LIN {X 0,Y 228.059,Z 101.561,A -85,B 0,C 180,E1 -19963.897,E2 -19963.897} C_VEL
LIN {X 0,Y 228.095,Z 101.553,A -85,B 0,C 180,E1 -19967.544,E2 -19967.544} C_VEL
LIN {X 0,Y 228.307,Z 101.501,A -85,B 0,C 180,E1 -19971.145,E2 -19971.145} C_VEL
LIN {X 0,Y 228.357,Z 101.52,A -85,B 0,C 180,E1 -19972.928,E2 -19972.928} C_VEL
LIN {X 0,Y 228.555,Z 101.482,A -85,B 0,C 180,E1 -19978.237,E2 -19978.237} C_VEL
LIN {X 0,Y 228.554,Z 101.479,A -85,B 0,C 180,E1 -19981.761,E2 -19981.761} C_VEL
LIN {X 0,Y 228.355,Z 101.523,A -85,B 0,C 180,E1 -19987.07,E2 -19987.07} C_VEL
LIN {X 0,Y 228.163,Z 101.521,A -85,B 0,C 180,E1 -19990.649,E2 -19990.649} C_VEL
LIN {X 0,Y 228.065,Z 101.576,A -85,B 0,C 180,E1 -19994.271,E2 -19994.271} C_VEL
LIN {X 0,Y 228.002,Z 101.548,A -85,B 0,C 180,E1 -19997.952,E2 -19997.952} C_VEL
LIN {X 0,Y 227.929,Z 101.59,A -85,B 0,C 180,E1 -20002.328,E2 -20002.328} C_VEL
LIN {X 0,Y 227.94,Z 101.56,A -85,B 0,C 180,E1 -20006.601,E2 -20006.601} C_VEL
LIN {X 0,Y 227.895,Z 101.596,A -85,B 0,C 180,E1 -20010.29,E2 -20010.29} C_VEL
LIN {X 0,Y 227.887,Z 101.574,A -85,B 0,C 180,E1 -20013.717,E2 -20013.717} C_VEL
LIN {X 0,Y 227.869,Z 101.603,A -85,B 0,C 180,E1 -20018.085,E2 -20018.085} C_VEL
LIN {X 0,Y 227.832,Z 101.602,A -85,B 0,C 180,E1 -20022.736,E2 -20022.736} C_VEL
LIN {X 0,Y 227.806,Z 101.544,A -85,B 0,C 180,E1 -20027.257,E2 -20027.257} C_VEL
LIN {X 0,Y 227.867,Z 101.603,A -85,B 0,C 180,E1 -20031.914,E2 -20031.914} C_VEL
LIN {X 0,Y 227.938,Z 101.91,A -85,B 0,C 180,E1 -20032.933,E2 -20032.933} C_VEL
LIN {X 0,Y 228.317,Z 103.201,A -85,B 0,C 180,E1 -20033.245,E2 -20033.245} C_VEL
LIN {X 0,Y 230.06,Z 105.866,A -85,B 0,C 180,E1 -20033.685,E2 -20033.685} C_VEL
LIN {X 0,Y 238.774,Z 120.975,A -85,B 0,C 180,E1 -20035.759,E2 -20035.759} C_VEL
LIN {X 0,Y 245.282,Z 133.413,A -85,B 0,C 180,E1 -20037.221,E2 -20037.221} C_VEL
LIN {X 0,Y 252.662,Z 147.165,A -85,B 0,C 180,E1 -20038.75,E2 -20038.75} C_VEL
LIN {X 0,Y 261.888,Z 160.593,A -85,B 0,C 180,E1 -20040.392,E2 -20040.392} C_VEL
LIN {X 0,Y 272.615,Z 173.13,A -85,B 0,C 180,E1 -20042.043,E2 -20042.043} C_VEL
LIN {X 0,Y 286.64,Z 187.221,A -85,B 0,C 180,E1 -20043.918,E2 -20043.918} C_VEL
LIN {X 0,Y 299.816,Z 198.41,A -85,B 0,C 180,E1 -20045.476,E2 -20045.476} C_VEL
LIN {X 0,Y 307.546,Z 204.743,A -85,B 0,C 180,E1 -20046.479,E2 -20046.479} C_VEL
LIN {X 0,Y 315.788,Z 211.095,A -85,B 0,C 180,E1 -20047.769,E2 -20047.769} C_VEL
LIN {X 0,Y 323.401,Z 216.756,A -85,B 0,C 180,E1 -20049.138,E2 -20049.138} C_VEL
LIN {X 0,Y 331.374,Z 222.775,A -85,B 0,C 180,E1 -20050.773,E2 -20050.773} C_VEL
LIN {X 0,Y 338.305,Z 227.474,A -85,B 0,C 180,E1 -20052.346,E2 -20052.346} C_VEL
LIN {X 0,Y 345.383,Z 232.65,A -85,B 0,C 180,E1 -20054.203,E2 -20054.203} C_VEL
LIN {X 0,Y 348.898,Z 235.005,A -85,B 0,C 180,E1 -20055.211,E2 -20055.211} C_VEL
LIN {X 0,Y 353.812,Z 237.864,A -85,B 0,C 180,E1 -20056.732,E2 -20056.732} C_VEL
LIN {X 0,Y 357.264,Z 240.175,A -85,B 0,C 180,E1 -20057.969,E2 -20057.969} C_VEL
LIN {X 0,Y 361.923,Z 243.575,A -85,B 0,C 180,E1 -20059.935,E2 -20059.935} C_VEL
LIN {X 0,Y 364.411,Z 245.128,A -85,B 0,C 180,E1 -20061.125,E2 -20061.125} C_VEL
LIN {X 0,Y 368.049,Z 247.051,A -85,B 0,C 180,E1 -20063.188,E2 -20063.188} C_VEL
LIN {X 0,Y 369.965,Z 247.87,A -85,B 0,C 180,E1 -20064.55,E2 -20064.55} C_VEL
LIN {X 0,Y 371.214,Z 248.393,A -85,B 0,C 180,E1 -20065.657,E2 -20065.657} C_VEL
LIN {X 0,Y 372.226,Z 248.63,A -85,B 0,C 180,E1 -20066.753,E2 -20066.753} C_VEL
LIN {X 0,Y 372.866,Z 248.985,A -85,B 0,C 180,E1 -20067.84,E2 -20067.84} C_VEL
LIN {X 0,Y 373.208,Z 249.303,A -85,B 0,C 180,E1 -20068.921,E2 -20068.921} C_VEL
LIN {X 0,Y 373.393,Z 249.209,A -85,B 0,C 180,E1 -20070,E2 -20070} C_VEL
LIN {X 0,Y 373.242,Z 249.205,A -85,B 0,C 180,E1 -20071.079,E2 -20071.079} C_VEL
LIN {X 0,Y 372.792,Z 248.918,A -85,B 0,C 180,E1 -20072.349,E2 -20072.349} C_VEL
LIN {X 0,Y 372.235,Z 248.604,A -85,B 0,C 180,E1 -20073.247,E2 -20073.247} C_VEL
LIN {X 0,Y 371.236,Z 248.342,A -85,B 0,C 180,E1 -20074.343,E2 -20074.343} C_VEL
LIN {X 0,Y 369.961,Z 247.901,A -85,B 0,C 180,E1 -20075.45,E2 -20075.45} C_VEL
LIN {X 0,Y 368.054,Z 247.054,A -85,B 0,C 180,E1 -20076.818,E2 -20076.818} C_VEL
LIN {X 0,Y 364.414,Z 245.128,A -85,B 0,C 180,E1 -20078.875,E2 -20078.875} C_VEL
LIN {X 0,Y 361.957,Z 243.542,A -85,B 0,C 180,E1 -20080.064,E2 -20080.064} C_VEL
LIN {X 0,Y 357.625,Z 240.46,A -85,B 0,C 180,E1 -20081.885,E2 -20081.885} C_VEL
LIN {X 0,Y 355.895,Z 239.071,A -85,B 0,C 180,E1 -20082.546,E2 -20082.546} C_VEL
LIN {X 0,Y 351.899,Z 236.864,A -85,B 0,C 180,E1 -20083.866,E2 -20083.866} C_VEL
LIN {X 0,Y 345.467,Z 232.643,A -85,B 0,C 180,E1 -20085.783,E2 -20085.783} C_VEL
LIN {X 0,Y 338.635,Z 227.695,A -85,B 0,C 180,E1 -20087.573,E2 -20087.573} C_VEL
LIN {X 0,Y 331.088,Z 222.551,A -85,B 0,C 180,E1 -20089.286,E2 -20089.286} C_VEL
LIN {X 0,Y 323.395,Z 216.791,A -85,B 0,C 180,E1 -20090.859,E2 -20090.859} C_VEL
LIN {X 0,Y 315.769,Z 211.081,A -85,B 0,C 180,E1 -20092.232,E2 -20092.232} C_VEL
LIN {X 0,Y 307.369,Z 204.614,A -85,B 0,C 180,E1 -20093.547,E2 -20093.547} C_VEL
LIN {X 0,Y 299.628,Z 198.281,A -85,B 0,C 180,E1 -20094.546,E2 -20094.546} C_VEL
LIN {X 0,Y 285.842,Z 186.494,A -85,B 0,C 180,E1 -20096.18,E2 -20096.18} C_VEL
LIN {X 0,Y 271.597,Z 172.061,A -85,B 0,C 180,E1 -20098.104,E2 -20098.104} C_VEL
LIN {X 0,Y 260.976,Z 159.397,A -85,B 0,C 180,E1 -20099.76,E2 -20099.76} C_VEL
LIN {X 0,Y 252.815,Z 147.338,A -85,B 0,C 180,E1 -20101.224,E2 -20101.224} C_VEL
LIN {X 0,Y 245.819,Z 134.485,A -85,B 0,C 180,E1 -20102.662,E2 -20102.662} C_VEL
LIN {X 0,Y 238.898,Z 121.153,A -85,B 0,C 180,E1 -20104.214,E2 -20104.214} C_VEL
LIN {X 0,Y 231.588,Z 108.563,A -85,B 0,C 180,E1 -20105.934,E2 -20105.934} C_VEL
LIN {X 0,Y 229.825,Z 105.609,A -85,B 0,C 180,E1 -20106.368,E2 -20106.368} C_VEL
LIN {X 0,Y 228.192,Z 102.895,A -85,B 0,C 180,E1 -20106.799,E2 -20106.799} C_VEL
LIN {X 0,Y 227.936,Z 101.844,A -85,B 0,C 180,E1 -20107.114,E2 -20107.114} C_VEL
LIN {X 0,Y 227.828,Z 101.552,A -85,B 0,C 180,E1 -20110.376,E2 -20110.376} C_VEL
LIN {X 0,Y 227.829,Z 101.581,A -85,B 0,C 180,E1 -20115.194,E2 -20115.194} C_VEL
LIN {X 0,Y 227.835,Z 101.584,A -85,B 0,C 180,E1 -20119.627,E2 -20119.627} C_VEL
LIN {X 0,Y 227.899,Z 101.579,A -85,B 0,C 180,E1 -20124.133,E2 -20124.133} C_VEL
LIN {X 0,Y 227.867,Z 101.601,A -85,B 0,C 180,E1 -20128.379,E2 -20128.379} C_VEL
LIN {X 0,Y 227.877,Z 101.566,A -85,B 0,C 180,E1 -20132.445,E2 -20132.445} C_VEL
LIN {X 0,Y 227.913,Z 101.595,A -85,B 0,C 180,E1 -20136.368,E2 -20136.368} C_VEL
LIN {X 0,Y 227.941,Z 101.553,A -85,B 0,C 180,E1 -20140.176,E2 -20140.176} C_VEL
LIN {X 0,Y 228.057,Z 101.568,A -85,B 0,C 180,E1 -20143.899,E2 -20143.899} C_VEL
LIN {X 0,Y 228.094,Z 101.554,A -85,B 0,C 180,E1 -20147.545,E2 -20147.545} C_VEL
LIN {X 0,Y 228.306,Z 101.504,A -85,B 0,C 180,E1 -20151.147,E2 -20151.147} C_VEL
LIN {X 0,Y 228.355,Z 101.523,A -85,B 0,C 180,E1 -20152.93,E2 -20152.93} C_VEL
LIN {X 0,Y 228.554,Z 101.479,A -85,B 0,C 180,E1 -20158.239,E2 -20158.239} C_VEL
LIN {X 0,Y 228.555,Z 101.482,A -85,B 0,C 180,E1 -20161.763,E2 -20161.763} C_VEL
LIN {X 0,Y 228.357,Z 101.52,A -85,B 0,C 180,E1 -20167.072,E2 -20167.072} C_VEL
LIN {X 0,Y 228.164,Z 101.52,A -85,B 0,C 180,E1 -20170.651,E2 -20170.651} C_VEL
LIN {X 0,Y 228.066,Z 101.573,A -85,B 0,C 180,E1 -20174.273,E2 -20174.273} C_VEL
LIN {X 0,Y 228.004,Z 101.542,A -85,B 0,C 180,E1 -20177.954,E2 -20177.954} C_VEL
LIN {X 0,Y 227.932,Z 101.589,A -85,B 0,C 180,E1 -20182.33,E2 -20182.33} C_VEL
LIN {X 0,Y 227.943,Z 101.557,A -85,B 0,C 180,E1 -20186.603,E2 -20186.603} C_VEL
LIN {X 0,Y 227.899,Z 101.596,A -85,B 0,C 180,E1 -20190.292,E2 -20190.292} C_VEL
LIN {X 0,Y 227.879,Z 101.572,A -85,B 0,C 180,E1 -20193.721,E2 -20193.721} C_VEL
LIN {X 0,Y 227.846,Z 101.601,A -85,B 0,C 180,E1 -20198.092,E2 -20198.092} C_VEL
LIN {X 0,Y 227.808,Z 101.61,A -85,B 0,C 180,E1 -20202.744,E2 -20202.744} C_VEL
LIN {X 0,Y 227.843,Z 101.602,A -85,B 0,C 180,E1 -20207.505,E2 -20207.505} C_VEL
LIN {X 0,Y 229.24,Z 107.256,A -85,B 0,C 180,E1 -20211.227,E2 -20211.227} C_VEL
LIN {X 0,Y 230.08,Z 111.007,A -85,B 0,C 180,E1 -20213.398,E2 -20213.398} C_VEL
LIN {X 0,Y 231.749,Z 114.816,A -85,B 0,C 180,E1 -20213.952,E2 -20213.952} C_VEL
LIN {X 0,Y 237.983,Z 127.674,A -85,B 0,C 180,E1 -20215.491,E2 -20215.491} C_VEL
LIN {X 0,Y 243.516,Z 140.613,A -85,B 0,C 180,E1 -20216.822,E2 -20216.822} C_VEL
LIN {X 0,Y 247.22,Z 160.789,A -85,B 0,C 180,E1 -20218.055,E2 -20218.055} C_VEL
LIN {X 0,Y 247.03,Z 164.678,A -85,B 0,C 180,E1 -20218.158,E2 -20218.158} C_VEL
LIN {X 0,Y 244.85,Z 170.983,A -85,B 0,C 180,E1 -20218.056,E2 -20218.056} C_VEL
LIN {X 0,Y 242.29,Z 177.323,A -85,B 0,C 180,E1 -20217.898,E2 -20217.898} C_VEL
LIN {X 0,Y 241.549,Z 181.312,A -85,B 0,C 180,E1 -20217.925,E2 -20217.925} C_VEL
LIN {X 0,Y 240.118,Z 217.09,A -85,B 0,C 180,E1 -20218.998,E2 -20218.998} C_VEL
LIN {X 0,Y 239.184,Z 227.774,A -85,B 0,C 180,E1 -20219.503,E2 -20219.503} C_VEL
LIN {X 0,Y 237.783,Z 238.307,A -85,B 0,C 180,E1 -20220.204,E2 -20220.204} C_VEL
LIN {X 0,Y 235.894,Z 250.119,A -85,B 0,C 180,E1 -20221.288,E2 -20221.288} C_VEL
LIN {X 0,Y 233.605,Z 261.513,A -85,B 0,C 180,E1 -20222.691,E2 -20222.691} C_VEL
LIN {X 0,Y 231.127,Z 271.803,A -85,B 0,C 180,E1 -20224.322,E2 -20224.322} C_VEL
LIN {X 0,Y 228.993,Z 280.33,A -85,B 0,C 180,E1 -20226.005,E2 -20226.005} C_VEL
LIN {X 0,Y 227.02,Z 287.546,A -85,B 0,C 180,E1 -20227.714,E2 -20227.714} C_VEL
LIN {X 0,Y 225.012,Z 295.126,A -85,B 0,C 180,E1 -20229.905,E2 -20229.905} C_VEL
LIN {X 0,Y 223.146,Z 301.441,A -85,B 0,C 180,E1 -20232.117,E2 -20232.117} C_VEL
LIN {X 0,Y 221.647,Z 306.704,A -85,B 0,C 180,E1 -20234.364,E2 -20234.364} C_VEL
LIN {X 0,Y 220.182,Z 311.833,A -85,B 0,C 180,E1 -20237.089,E2 -20237.089} C_VEL
LIN {X 0,Y 219.312,Z 315.826,A -85,B 0,C 180,E1 -20239.849,E2 -20239.849} C_VEL
LIN {X 0,Y 218.737,Z 318.78,A -85,B 0,C 180,E1 -20242.616,E2 -20242.616} C_VEL
LIN {X 0,Y 218.501,Z 321.234,A -85,B 0,C 180,E1 -20246.312,E2 -20246.312} C_VEL
LIN {X 0,Y 218.524,Z 321.827,A -85,B 0,C 180,E1 -20248.157,E2 -20248.157} C_VEL
LIN {X 0,Y 218.629,Z 321.985,A -85,B 0,C 180,E1 -20250,E2 -20250} C_VEL
LIN {X 0,Y 218.524,Z 321.827,A -85,B 0,C 180,E1 -20251.843,E2 -20251.843} C_VEL
LIN {X 0,Y 218.484,Z 320.97,A -85,B 0,C 180,E1 -20254.292,E2 -20254.292} C_VEL
LIN {X 0,Y 218.737,Z 318.78,A -85,B 0,C 180,E1 -20257.384,E2 -20257.384} C_VEL
LIN {X 0,Y 219.312,Z 315.826,A -85,B 0,C 180,E1 -20260.151,E2 -20260.151} C_VEL
LIN {X 0,Y 220.182,Z 311.833,A -85,B 0,C 180,E1 -20262.911,E2 -20262.911} C_VEL
LIN {X 0,Y 221.647,Z 306.704,A -85,B 0,C 180,E1 -20265.636,E2 -20265.636} C_VEL
LIN {X 0,Y 223.15,Z 301.441,A -85,B 0,C 180,E1 -20267.883,E2 -20267.883} C_VEL
LIN {X 0,Y 225.051,Z 295.127,A -85,B 0,C 180,E1 -20270.091,E2 -20270.091} C_VEL
LIN {X 0,Y 226.622,Z 289.174,A -85,B 0,C 180,E1 -20271.848,E2 -20271.848} C_VEL
LIN {X 0,Y 228.472,Z 282.248,A -85,B 0,C 180,E1 -20273.571,E2 -20273.571} C_VEL
LIN {X 0,Y 230.659,Z 274.074,A -85,B 0,C 180,E1 -20275.25,E2 -20275.25} C_VEL
LIN {X 0,Y 232.669,Z 265.565,A -85,B 0,C 180,E1 -20276.7,E2 -20276.7} C_VEL
LIN {X 0,Y 234.586,Z 256.854,A -85,B 0,C 180,E1 -20277.912,E2 -20277.912} C_VEL
LIN {X 0,Y 236.222,Z 248.105,A -85,B 0,C 180,E1 -20278.912,E2 -20278.912} C_VEL
LIN {X 0,Y 237.81,Z 238.308,A -85,B 0,C 180,E1 -20279.792,E2 -20279.792} C_VEL
LIN {X 0,Y 239.138,Z 227.8,A -85,B 0,C 180,E1 -20280.502,E2 -20280.502} C_VEL
LIN {X 0,Y 240.011,Z 218.263,A -85,B 0,C 180,E1 -20280.96,E2 -20280.96} C_VEL
LIN {X 0,Y 241.305,Z 187.828,A -85,B 0,C 180,E1 -20281.887,E2 -20281.887} C_VEL
LIN {X 0,Y 241.985,Z 166.994,A -85,B 0,C 180,E1 -20282.502,E2 -20282.502} C_VEL
LIN {X 0,Y 238.111,Z 144.56,A -85,B 0,C 180,E1 -20283.887,E2 -20283.887} C_VEL
LIN {X 0,Y 234.794,Z 136.065,A -85,B 0,C 180,E1 -20284.736,E2 -20284.736} C_VEL
LIN {X 0,Y 228.627,Z 122.664,A -85,B 0,C 180,E1 -20286.316,E2 -20286.316} C_VEL
LIN {X 0,Y 224.217,Z 114.028,A -85,B 0,C 180,E1 -20287.483,E2 -20287.483} C_VEL
LIN {X 0,Y 222.783,Z 110.774,A -85,B 0,C 180,E1 -20288.007,E2 -20288.007} C_VEL
LIN {X 0,Y 221.489,Z 105.488,A -85,B 0,C 180,E1 -20291.331,E2 -20291.331} C_VEL
LIN {X 0,Y 220.777,Z 102.498,A -85,B 0,C 180,E1 -20293.48,E2 -20293.48} C_VEL
LIN {X 0,Y 220.769,Z 102.48,A -85,B 0,C 180,E1 -20298.046,E2 -20298.046} C_VEL
LIN {X 0,Y 220.808,Z 102.462,A -85,B 0,C 180,E1 -20300.462,E2 -20300.462} C_VEL
LIN {X 0,Y 220.803,Z 102.454,A -85,B 0,C 180,E1 -20305.044,E2 -20305.044} C_VEL
LIN {X 0,Y 220.836,Z 102.477,A -85,B 0,C 180,E1 -20309.389,E2 -20309.389} C_VEL
LIN {X 0,Y 220.896,Z 102.434,A -85,B 0,C 180,E1 -20313.549,E2 -20313.549} C_VEL
LIN {X 0,Y 220.88,Z 102.468,A -85,B 0,C 180,E1 -20317.553,E2 -20317.553} C_VEL
LIN {X 0,Y 220.986,Z 102.42,A -85,B 0,C 180,E1 -20322.57,E2 -20322.57} C_VEL
LIN {X 0,Y 221.028,Z 102.44,A -85,B 0,C 180,E1 -20327.138,E2 -20327.138} C_VEL
LIN {X 0,Y 221.238,Z 102.379,A -85,B 0,C 180,E1 -20330.86,E2 -20330.86} C_VEL
LIN {X 0,Y 221.292,Z 102.396,A -85,B 0,C 180,E1 -20332.701,E2 -20332.701} C_VEL
LIN {X 0,Y 221.513,Z 102.358,A -85,B 0,C 180,E1 -20338.181,E2 -20338.181} C_VEL
LIN {X 0,Y 221.512,Z 102.356,A -85,B 0,C 180,E1 -20341.817,E2 -20341.817} C_VEL
LIN {X 0,Y 221.29,Z 102.399,A -85,B 0,C 180,E1 -20347.297,E2 -20347.297} C_VEL
LIN {X 0,Y 221.112,Z 102.401,A -85,B 0,C 180,E1 -20350.993,E2 -20350.993} C_VEL
LIN {X 0,Y 221.016,Z 102.435,A -85,B 0,C 180,E1 -20356.629,E2 -20356.629} C_VEL
LIN {X 0,Y 220.891,Z 102.437,A -85,B 0,C 180,E1 -20360.485,E2 -20360.485} C_VEL
LIN {X 0,Y 220.866,Z 102.467,A -85,B 0,C 180,E1 -20364.434,E2 -20364.434} C_VEL
LIN {X 0,Y 220.825,Z 102.45,A -85,B 0,C 180,E1 -20368.514,E2 -20368.514} C_VEL
LIN {X 0,Y 220.821,Z 102.464,A -85,B 0,C 180,E1 -20372.754,E2 -20372.754} C_VEL
LIN {X 0,Y 220.836,Z 102.478,A -85,B 0,C 180,E1 -20377.287,E2 -20377.287} C_VEL
LIN {X 0,Y 220.784,Z 102.469,A -85,B 0,C 180,E1 -20381.948,E2 -20381.948} C_VEL
LIN {X 0,Y 220.768,Z 102.441,A -85,B 0,C 180,E1 -20385.545,E2 -20385.545} C_VEL
LIN {X 0,Y 220.806,Z 102.44,A -85,B 0,C 180,E1 -20390.463,E2 -20390.463} C_VEL
LIN {X 0,Y 220.874,Z 102.767,A -85,B 0,C 180,E1 -20391.554,E2 -20391.554} C_VEL
LIN {X 0,Y 221.235,Z 104.073,A -85,B 0,C 180,E1 -20391.889,E2 -20391.889} C_VEL
LIN {X 0,Y 222.818,Z 106.604,A -85,B 0,C 180,E1 -20392.324,E2 -20392.324} C_VEL
LIN {X 0,Y 228.374,Z 115.616,A -85,B 0,C 180,E1 -20393.745,E2 -20393.745} C_VEL
LIN {X 0,Y 236.785,Z 130.683,A -85,B 0,C 180,E1 -20395.779,E2 -20395.779} C_VEL
LIN {X 0,Y 246.3,Z 149.277,A -85,B 0,C 180,E1 -20397.912,E2 -20397.912} C_VEL
LIN {X 0,Y 254.449,Z 161.727,A -85,B 0,C 180,E1 -20399.465,E2 -20399.465} C_VEL
LIN {X 0,Y 261.832,Z 171.211,A -85,B 0,C 180,E1 -20400.713,E2 -20400.713} C_VEL
LIN {X 0,Y 273.471,Z 184.014,A -85,B 0,C 180,E1 -20402.455,E2 -20402.455} C_VEL
LIN {X 0,Y 285.366,Z 195.325,A -85,B 0,C 180,E1 -20404.015,E2 -20404.015} C_VEL
LIN {X 0,Y 297.064,Z 205.177,A -85,B 0,C 180,E1 -20405.415,E2 -20405.415} C_VEL
LIN {X 0,Y 305.278,Z 211.84,A -85,B 0,C 180,E1 -20406.528,E2 -20406.528} C_VEL
LIN {X 0,Y 313.149,Z 217.956,A -85,B 0,C 180,E1 -20407.782,E2 -20407.782} C_VEL
LIN {X 0,Y 321.079,Z 223.725,A -85,B 0,C 180,E1 -20409.211,E2 -20409.211} C_VEL
LIN {X 0,Y 329.305,Z 229.918,A -85,B 0,C 180,E1 -20410.923,E2 -20410.923} C_VEL
LIN {X 0,Y 335.922,Z 234.284,A -85,B 0,C 180,E1 -20412.435,E2 -20412.435} C_VEL
LIN {X 0,Y 343.051,Z 239.531,A -85,B 0,C 180,E1 -20414.337,E2 -20414.337} C_VEL
LIN {X 0,Y 348.672,Z 243.15,A -85,B 0,C 180,E1 -20416.003,E2 -20416.003} C_VEL
LIN {X 0,Y 352.897,Z 245.512,A -85,B 0,C 180,E1 -20417.377,E2 -20417.377} C_VEL
LIN {X 0,Y 357.62,Z 249.055,A -85,B 0,C 180,E1 -20419.294,E2 -20419.294} C_VEL
LIN {X 0,Y 361.346,Z 251.519,A -85,B 0,C 180,E1 -20421.049,E2 -20421.049} C_VEL
LIN {X 0,Y 363.544,Z 252.704,A -85,B 0,C 180,E1 -20422.223,E2 -20422.223} C_VEL
LIN {X 0,Y 365.419,Z 253.659,A -85,B 0,C 180,E1 -20423.374,E2 -20423.374} C_VEL
LIN {X 0,Y 367.1,Z 254.352,A -85,B 0,C 180,E1 -20424.568,E2 -20424.568} C_VEL
LIN {X 0,Y 368.285,Z 254.845,A -85,B 0,C 180,E1 -20425.622,E2 -20425.622} C_VEL
LIN {X 0,Y 369.316,Z 255.107,A -85,B 0,C 180,E1 -20426.727,E2 -20426.727} C_VEL
LIN {X 0,Y 369.972,Z 255.445,A -85,B 0,C 180,E1 -20427.823,E2 -20427.823} C_VEL
LIN {X 0,Y 370.311,Z 255.754,A -85,B 0,C 180,E1 -20428.913,E2 -20428.913} C_VEL
LIN {X 0,Y 370.495,Z 255.693,A -85,B 0,C 180,E1 -20430,E2 -20430} C_VEL
LIN {X 0,Y 370.339,Z 255.679,A -85,B 0,C 180,E1 -20431.087,E2 -20431.087} C_VEL
LIN {X 0,Y 369.975,Z 255.415,A -85,B 0,C 180,E1 -20432.177,E2 -20432.177} C_VEL
LIN {X 0,Y 369.326,Z 255.057,A -85,B 0,C 180,E1 -20433.273,E2 -20433.273} C_VEL
LIN {X 0,Y 368.296,Z 254.797,A -85,B 0,C 180,E1 -20434.378,E2 -20434.378} C_VEL
LIN {X 0,Y 366.999,Z 254.346,A -85,B 0,C 180,E1 -20435.494,E2 -20435.494} C_VEL
LIN {X 0,Y 365.433,Z 253.638,A -85,B 0,C 180,E1 -20436.626,E2 -20436.626} C_VEL
LIN {X 0,Y 362.338,Z 252.068,A -85,B 0,C 180,E1 -20438.43,E2 -20438.43} C_VEL
LIN {X 0,Y 358.862,Z 249.906,A -85,B 0,C 180,E1 -20440.152,E2 -20440.152} C_VEL
LIN {X 0,Y 354.957,Z 247.125,A -85,B 0,C 180,E1 -20441.812,E2 -20441.812} C_VEL
LIN {X 0,Y 352.801,Z 245.433,A -85,B 0,C 180,E1 -20442.658,E2 -20442.658} C_VEL
LIN {X 0,Y 347.99,Z 242.708,A -85,B 0,C 180,E1 -20444.212,E2 -20444.212} C_VEL
LIN {X 0,Y 343.044,Z 239.539,A -85,B 0,C 180,E1 -20445.66,E2 -20445.66} C_VEL
LIN {X 0,Y 338.086,Z 235.936,A -85,B 0,C 180,E1 -20447.017,E2 -20447.017} C_VEL
LIN {X 0,Y 330.721,Z 230.874,A -85,B 0,C 180,E1 -20448.764,E2 -20448.764} C_VEL
LIN {X 0,Y 323.251,Z 225.325,A -85,B 0,C 180,E1 -20450.357,E2 -20450.357} C_VEL
LIN {X 0,Y 314.811,Z 219.201,A -85,B 0,C 180,E1 -20451.933,E2 -20451.933} C_VEL
LIN {X 0,Y 306.362,Z 212.683,A -85,B 0,C 180,E1 -20453.309,E2 -20453.309} C_VEL
LIN {X 0,Y 298.371,Z 206.277,A -85,B 0,C 180,E1 -20454.423,E2 -20454.423} C_VEL
LIN {X 0,Y 286.875,Z 196.615,A -85,B 0,C 180,E1 -20455.802,E2 -20455.802} C_VEL
LIN {X 0,Y 276.959,Z 187.471,A -85,B 0,C 180,E1 -20457.067,E2 -20457.067} C_VEL
LIN {X 0,Y 264.203,Z 174.057,A -85,B 0,C 180,E1 -20458.91,E2 -20458.91} C_VEL
LIN {X 0,Y 254.983,Z 162.535,A -85,B 0,C 180,E1 -20460.438,E2 -20460.438} C_VEL
LIN {X 0,Y 246.306,Z 149.26,A -85,B 0,C 180,E1 -20462.088,E2 -20462.088} C_VEL
LIN {X 0,Y 239.106,Z 135.314,A -85,B 0,C 180,E1 -20463.677,E2 -20463.677} C_VEL
LIN {X 0,Y 231.131,Z 120.328,A -85,B 0,C 180,E1 -20465.575,E2 -20465.575} C_VEL
LIN {X 0,Y 224.994,Z 110.1,A -85,B 0,C 180,E1 -20467.109,E2 -20467.109} C_VEL
LIN {X 0,Y 222.657,Z 106.438,A -85,B 0,C 180,E1 -20467.715,E2 -20467.715} C_VEL
LIN {X 0,Y 221.06,Z 103.617,A -85,B 0,C 180,E1 -20468.184,E2 -20468.184} C_VEL
LIN {X 0,Y 220.857,Z 102.683,A -85,B 0,C 180,E1 -20468.516,E2 -20468.516} C_VEL
LIN {X 0,Y 220.768,Z 102.418,A -85,B 0,C 180,E1 -20471.953,E2 -20471.953} C_VEL
LIN {X 0,Y 220.773,Z 102.467,A -85,B 0,C 180,E1 -20475.547,E2 -20475.547} C_VEL
LIN {X 0,Y 220.808,Z 102.464,A -85,B 0,C 180,E1 -20480.465,E2 -20480.465} C_VEL
LIN {X 0,Y 220.832,Z 102.477,A -85,B 0,C 180,E1 -20482.796,E2 -20482.796} C_VEL
LIN {X 0,Y 220.821,Z 102.464,A -85,B 0,C 180,E1 -20487.246,E2 -20487.246} C_VEL
LIN {X 0,Y 220.825,Z 102.45,A -85,B 0,C 180,E1 -20491.486,E2 -20491.486} C_VEL
LIN {X 0,Y 220.866,Z 102.467,A -85,B 0,C 180,E1 -20495.566,E2 -20495.566} C_VEL
LIN {X 0,Y 220.891,Z 102.437,A -85,B 0,C 180,E1 -20499.515,E2 -20499.515} C_VEL
LIN {X 0,Y 221.016,Z 102.435,A -85,B 0,C 180,E1 -20503.371,E2 -20503.371} C_VEL
LIN {X 0,Y 221.112,Z 102.401,A -85,B 0,C 180,E1 -20509.007,E2 -20509.007} C_VEL
LIN {X 0,Y 221.29,Z 102.399,A -85,B 0,C 180,E1 -20512.703,E2 -20512.703} C_VEL
LIN {X 0,Y 221.512,Z 102.356,A -85,B 0,C 180,E1 -20518.183,E2 -20518.183} C_VEL
LIN {X 0,Y 221.513,Z 102.358,A -85,B 0,C 180,E1 -20521.819,E2 -20521.819} C_VEL
LIN {X 0,Y 221.292,Z 102.396,A -85,B 0,C 180,E1 -20527.299,E2 -20527.299} C_VEL
LIN {X 0,Y 221.113,Z 102.4,A -85,B 0,C 180,E1 -20530.995,E2 -20530.995} C_VEL
LIN {X 0,Y 221.018,Z 102.428,A -85,B 0,C 180,E1 -20536.631,E2 -20536.631} C_VEL
LIN {X 0,Y 220.894,Z 102.436,A -85,B 0,C 180,E1 -20540.487,E2 -20540.487} C_VEL
LIN {X 0,Y 220.869,Z 102.461,A -85,B 0,C 180,E1 -20544.436,E2 -20544.436} C_VEL
LIN {X 0,Y 220.829,Z 102.451,A -85,B 0,C 180,E1 -20548.516,E2 -20548.516} C_VEL
LIN {X 0,Y 220.818,Z 102.459,A -85,B 0,C 180,E1 -20552.757,E2 -20552.757} C_VEL
LIN {X 0,Y 220.813,Z 102.481,A -85,B 0,C 180,E1 -20557.279,E2 -20557.279} C_VEL
LIN {X 0,Y 220.796,Z 102.462,A -85,B 0,C 180,E1 -20560.189,E2 -20560.189} C_VEL
LIN {X 0,Y 220.77,Z 102.472,A -85,B 0,C 180,E1 -20564.456,E2 -20564.456} C_VEL
LIN {X 0,Y 220.78,Z 102.537,A -85,B 0,C 180,E1 -20566.645,E2 -20566.645} C_VEL
LIN {X 0,Y 222.642,Z 110.068,A -85,B 0,C 180,E1 -20571.654,E2 -20571.654} C_VEL
LIN {X 0,Y 222.97,Z 111.311,A -85,B 0,C 180,E1 -20572.126,E2 -20572.126} C_VEL
LIN {X 0,Y 229.659,Z 124.833,A -85,B 0,C 180,E1 -20573.953,E2 -20573.953} C_VEL
LIN {X 0,Y 236.147,Z 139.24,A -85,B 0,C 180,E1 -20575.604,E2 -20575.604} C_VEL
LIN {X 0,Y 238.114,Z 144.509,A -85,B 0,C 180,E1 -20576.112,E2 -20576.112} C_VEL
LIN {X 0,Y 241.448,Z 163.621,A -85,B 0,C 180,E1 -20577.301,E2 -20577.301} C_VEL
LIN {X 0,Y 242.072,Z 168.246,A -85,B 0,C 180,E1 -20577.554,E2 -20577.554} C_VEL
LIN {X 0,Y 241.549,Z 181.312,A -85,B 0,C 180,E1 -20577.925,E2 -20577.925} C_VEL
LIN {X 0,Y 240.728,Z 187.162,A -85,B 0,C 180,E1 -20577.999,E2 -20577.999} C_VEL
LIN {X 0,Y 235.124,Z 206.176,A -85,B 0,C 180,E1 -20577.802,E2 -20577.802} C_VEL
LIN {X 0,Y 234.34,Z 212.004,A -85,B 0,C 180,E1 -20577.916,E2 -20577.916} C_VEL
LIN {X 0,Y 233.375,Z 224.851,A -85,B 0,C 180,E1 -20578.461,E2 -20578.461} C_VEL
LIN {X 0,Y 232.06,Z 235.543,A -85,B 0,C 180,E1 -20579.139,E2 -20579.139} C_VEL
LIN {X 0,Y 230.563,Z 244.895,A -85,B 0,C 180,E1 -20579.931,E2 -20579.931} C_VEL
LIN {X 0,Y 228.635,Z 255.031,A -85,B 0,C 180,E1 -20581.044,E2 -20581.044} C_VEL
LIN {X 0,Y 226.646,Z 264.023,A -85,B 0,C 180,E1 -20582.281,E2 -20582.281} C_VEL
LIN {X 0,Y 224.461,Z 272.747,A -85,B 0,C 180,E1 -20583.752,E2 -20583.752} C_VEL
LIN {X 0,Y 222.496,Z 280.139,A -85,B 0,C 180,E1 -20585.258,E2 -20585.258} C_VEL
LIN {X 0,Y 220.429,Z 287.355,A -85,B 0,C 180,E1 -20587.01,E2 -20587.01} C_VEL
LIN {X 0,Y 218.323,Z 294.935,A -85,B 0,C 180,E1 -20589.262,E2 -20589.262} C_VEL
LIN {X 0,Y 216.352,Z 301.249,A -85,B 0,C 180,E1 -20591.535,E2 -20591.535} C_VEL
LIN {X 0,Y 214.779,Z 306.512,A -85,B 0,C 180,E1 -20593.851,E2 -20593.851} C_VEL
LIN {X 0,Y 213.221,Z 311.641,A -85,B 0,C 180,E1 -20596.66,E2 -20596.66} C_VEL
LIN {X 0,Y 212.298,Z 315.635,A -85,B 0,C 180,E1 -20599.509,E2 -20599.509} C_VEL
LIN {X 0,Y 211.671,Z 318.589,A -85,B 0,C 180,E1 -20602.368,E2 -20602.368} C_VEL
LIN {X 0,Y 211.42,Z 321.044,A -85,B 0,C 180,E1 -20606.188,E2 -20606.188} C_VEL
LIN {X 0,Y 211.426,Z 321.636,A -85,B 0,C 180,E1 -20608.095,E2 -20608.095} C_VEL
LIN {X 0,Y 211.545,Z 321.795,A -85,B 0,C 180,E1 -20610,E2 -20610} C_VEL
LIN {X 0,Y 211.426,Z 321.636,A -85,B 0,C 180,E1 -20611.905,E2 -20611.905} C_VEL
LIN {X 0,Y 211.396,Z 320.927,A -85,B 0,C 180,E1 -20614.145,E2 -20614.145} C_VEL
LIN {X 0,Y 211.671,Z 318.589,A -85,B 0,C 180,E1 -20617.632,E2 -20617.632} C_VEL
LIN {X 0,Y 212.298,Z 315.635,A -85,B 0,C 180,E1 -20620.491,E2 -20620.491} C_VEL
LIN {X 0,Y 213.22,Z 311.641,A -85,B 0,C 180,E1 -20623.34,E2 -20623.34} C_VEL
LIN {X 0,Y 214.78,Z 306.512,A -85,B 0,C 180,E1 -20626.149,E2 -20626.149} C_VEL
LIN {X 0,Y 216.357,Z 301.249,A -85,B 0,C 180,E1 -20628.464,E2 -20628.464} C_VEL
LIN {X 0,Y 218.364,Z 294.936,A -85,B 0,C 180,E1 -20630.734,E2 -20630.734} C_VEL
LIN {X 0,Y 220.012,Z 288.983,A -85,B 0,C 180,E1 -20632.54,E2 -20632.54} C_VEL
LIN {X 0,Y 221.978,Z 282.058,A -85,B 0,C 180,E1 -20634.305,E2 -20634.305} C_VEL
LIN {X 0,Y 224.246,Z 273.883,A -85,B 0,C 180,E1 -20636.025,E2 -20636.025} C_VEL
LIN {X 0,Y 226.338,Z 265.375,A -85,B 0,C 180,E1 -20637.509,E2 -20637.509} C_VEL
LIN {X 0,Y 228.331,Z 256.664,A -85,B 0,C 180,E1 -20638.746,E2 -20638.746} C_VEL
LIN {X 0,Y 230.044,Z 247.915,A -85,B 0,C 180,E1 -20639.765,E2 -20639.765} C_VEL
LIN {X 0,Y 231.674,Z 238.117,A -85,B 0,C 180,E1 -20640.665,E2 -20640.665} C_VEL
LIN {X 0,Y 233.033,Z 227.816,A -85,B 0,C 180,E1 -20641.375,E2 -20641.375} C_VEL
LIN {X 0,Y 233.975,Z 217.608,A -85,B 0,C 180,E1 -20641.873,E2 -20641.873} C_VEL
LIN {X 0,Y 235.665,Z 178.995,A -85,B 0,C 180,E1 -20643.052,E2 -20643.052} C_VEL
LIN {X 0,Y 235.976,Z 168.123,A -85,B 0,C 180,E1 -20643.389,E2 -20643.389} C_VEL
LIN {X 0,Y 232.45,Z 147.092,A -85,B 0,C 180,E1 -20644.729,E2 -20644.729} C_VEL
LIN {X 0,Y 228.078,Z 136.184,A -85,B 0,C 180,E1 -20645.902,E2 -20645.902} C_VEL
LIN {X 0,Y 221.785,Z 122.942,A -85,B 0,C 180,E1 -20647.606,E2 -20647.606} C_VEL
LIN {X 0,Y 217.168,Z 114.145,A -85,B 0,C 180,E1 -20648.908,E2 -20648.908} C_VEL
LIN {X 0,Y 215.508,Z 110.625,A -85,B 0,C 180,E1 -20649.508,E2 -20649.508} C_VEL
LIN {X 0,Y 213.928,Z 104.35,A -85,B 0,C 180,E1 -20653.717,E2 -20653.717} C_VEL
LIN {X 0,Y 213.744,Z 103.351,A -85,B 0,C 180,E1 -20654.679,E2 -20654.679} C_VEL
LIN {X 0,Y 213.718,Z 103.346,A -85,B 0,C 180,E1 -20659.142,E2 -20659.142} C_VEL
LIN {X 0,Y 213.746,Z 103.348,A -85,B 0,C 180,E1 -20663.711,E2 -20663.711} C_VEL
LIN {X 0,Y 213.769,Z 103.352,A -85,B 0,C 180,E1 -20668.262,E2 -20668.262} C_VEL
LIN {X 0,Y 213.828,Z 103.313,A -85,B 0,C 180,E1 -20672.602,E2 -20672.602} C_VEL
LIN {X 0,Y 213.854,Z 103.345,A -85,B 0,C 180,E1 -20676.952,E2 -20676.952} C_VEL
LIN {X 0,Y 213.945,Z 103.299,A -85,B 0,C 180,E1 -20682.803,E2 -20682.803} C_VEL
LIN {X 0,Y 213.982,Z 103.322,A -85,B 0,C 180,E1 -20686.707,E2 -20686.707} C_VEL
LIN {X 0,Y 214.169,Z 103.258,A -85,B 0,C 180,E1 -20690.555,E2 -20690.555} C_VEL
LIN {X 0,Y 214.229,Z 103.269,A -85,B 0,C 180,E1 -20692.459,E2 -20692.459} C_VEL
LIN {X 0,Y 214.446,Z 103.238,A -85,B 0,C 180,E1 -20698.121,E2 -20698.121} C_VEL
LIN {X 0,Y 214.547,Z 103.21,A -85,B 0,C 180,E1 -20699.999,E2 -20699.999} C_VEL
LIN {X 0,Y 214.446,Z 103.235,A -85,B 0,C 180,E1 -20701.877,E2 -20701.877} C_VEL
LIN {X 0,Y 214.228,Z 103.273,A -85,B 0,C 180,E1 -20707.539,E2 -20707.539} C_VEL
LIN {X 0,Y 214.045,Z 103.284,A -85,B 0,C 180,E1 -20711.361,E2 -20711.361} C_VEL
LIN {X 0,Y 213.934,Z 103.334,A -85,B 0,C 180,E1 -20715.236,E2 -20715.236} C_VEL
LIN {X 0,Y 213.838,Z 103.306,A -85,B 0,C 180,E1 -20719.186,E2 -20719.186} C_VEL
LIN {X 0,Y 213.846,Z 103.349,A -85,B 0,C 180,E1 -20723.226,E2 -20723.226} C_VEL
LIN {X 0,Y 213.827,Z 103.315,A -85,B 0,C 180,E1 -20727.449,E2 -20727.449} C_VEL
LIN {X 0,Y 213.768,Z 103.356,A -85,B 0,C 180,E1 -20731.736,E2 -20731.736} C_VEL
LIN {X 0,Y 213.752,Z 103.345,A -85,B 0,C 180,E1 -20736.285,E2 -20736.285} C_VEL
LIN {X 0,Y 213.721,Z 103.342,A -85,B 0,C 180,E1 -20741.122,E2 -20741.122} C_VEL
LIN {X 0,Y 213.727,Z 103.361,A -85,B 0,C 180,E1 -20743.672,E2 -20743.672} C_VEL
LIN {X 0,Y 213.7,Z 103.307,A -85,B 0,C 180,E1 -20746.344,E2 -20746.344} C_VEL
LIN {X 0,Y 213.794,Z 103.502,A -85,B 0,C 180,E1 -20749.96,E2 -20749.96} C_VEL
LIN {X 0,Y 214.063,Z 104.635,A -85,B 0,C 180,E1 -20750.372,E2 -20750.372} C_VEL
LIN {X 0,Y 215.627,Z 107.296,A -85,B 0,C 180,E1 -20750.852,E2 -20750.852} C_VEL
LIN {X 0,Y 216.547,Z 108.567,A -85,B 0,C 180,E1 -20751.104,E2 -20751.104} C_VEL
LIN {X 0,Y 223.568,Z 119.926,A -85,B 0,C 180,E1 -20753.001,E2 -20753.001} C_VEL
LIN {X 0,Y 231.862,Z 134.971,A -85,B 0,C 180,E1 -20755.1,E2 -20755.1} C_VEL
LIN {X 0,Y 241.207,Z 153.46,A -85,B 0,C 180,E1 -20757.29,E2 -20757.29} C_VEL
LIN {X 0,Y 249.984,Z 167.005,A -85,B 0,C 180,E1 -20759.028,E2 -20759.028} C_VEL
LIN {X 0,Y 259.189,Z 178.625,A -85,B 0,C 180,E1 -20760.614,E2 -20760.614} C_VEL
LIN {X 0,Y 271.317,Z 191.6,A -85,B 0,C 180,E1 -20762.438,E2 -20762.438} C_VEL
LIN {X 0,Y 282.411,Z 202.002,A -85,B 0,C 180,E1 -20763.923,E2 -20763.923} C_VEL
LIN {X 0,Y 292.263,Z 210.35,A -85,B 0,C 180,E1 -20765.196,E2 -20765.196} C_VEL
LIN {X 0,Y 301.379,Z 217.746,A -85,B 0,C 180,E1 -20766.443,E2 -20766.443} C_VEL
LIN {X 0,Y 308.36,Z 223.145,A -85,B 0,C 180,E1 -20767.534,E2 -20767.534} C_VEL
LIN {X 0,Y 316.304,Z 228.978,A -85,B 0,C 180,E1 -20768.937,E2 -20768.937} C_VEL
LIN {X 0,Y 323.612,Z 234.482,A -85,B 0,C 180,E1 -20770.412,E2 -20770.412} C_VEL
LIN {X 0,Y 330.772,Z 239.383,A -85,B 0,C 180,E1 -20772.006,E2 -20772.006} C_VEL
LIN {X 0,Y 337.806,Z 244.516,A -85,B 0,C 180,E1 -20773.817,E2 -20773.817} C_VEL
LIN {X 0,Y 344.802,Z 249.073,A -85,B 0,C 180,E1 -20775.842,E2 -20775.842} C_VEL
LIN {X 0,Y 349.042,Z 251.434,A -85,B 0,C 180,E1 -20777.204,E2 -20777.204} C_VEL
LIN {X 0,Y 353.971,Z 255.109,A -85,B 0,C 180,E1 -20779.182,E2 -20779.182} C_VEL
LIN {X 0,Y 357.757,Z 257.617,A -85,B 0,C 180,E1 -20780.958,E2 -20780.958} C_VEL
LIN {X 0,Y 361.218,Z 259.483,A -85,B 0,C 180,E1 -20782.868,E2 -20782.868} C_VEL
LIN {X 0,Y 363.568,Z 260.516,A -85,B 0,C 180,E1 -20784.454,E2 -20784.454} C_VEL
LIN {X 0,Y 364.895,Z 261.068,A -85,B 0,C 180,E1 -20785.581,E2 -20785.581} C_VEL
LIN {X 0,Y 366.034,Z 261.398,A -85,B 0,C 180,E1 -20786.766,E2 -20786.766} C_VEL
LIN {X 0,Y 366.653,Z 261.715,A -85,B 0,C 180,E1 -20787.803,E2 -20787.803} C_VEL
LIN {X 0,Y 366.993,Z 262.021,A -85,B 0,C 180,E1 -20788.903,E2 -20788.903} C_VEL
LIN {X 0,Y 367.193,Z 261.964,A -85,B 0,C 180,E1 -20790,E2 -20790} C_VEL
LIN {X 0,Y 367.026,Z 261.949,A -85,B 0,C 180,E1 -20791.097,E2 -20791.097} C_VEL
LIN {X 0,Y 366.659,Z 261.683,A -85,B 0,C 180,E1 -20792.197,E2 -20792.197} C_VEL
LIN {X 0,Y 365.982,Z 261.335,A -85,B 0,C 180,E1 -20793.303,E2 -20793.303} C_VEL
LIN {X 0,Y 364.893,Z 261.042,A -85,B 0,C 180,E1 -20794.419,E2 -20794.419} C_VEL
LIN {X 0,Y 363.54,Z 260.529,A -85,B 0,C 180,E1 -20795.547,E2 -20795.547} C_VEL
LIN {X 0,Y 361.227,Z 259.479,A -85,B 0,C 180,E1 -20797.144,E2 -20797.144} C_VEL
LIN {X 0,Y 357.751,Z 257.601,A -85,B 0,C 180,E1 -20799.042,E2 -20799.042} C_VEL
LIN {X 0,Y 355.228,Z 255.977,A -85,B 0,C 180,E1 -20800.257,E2 -20800.257} C_VEL
LIN {X 0,Y 351.742,Z 253.523,A -85,B 0,C 180,E1 -20801.753,E2 -20801.753} C_VEL
LIN {X 0,Y 349.05,Z 251.469,A -85,B 0,C 180,E1 -20802.796,E2 -20802.796} C_VEL
LIN {X 0,Y 344.788,Z 249.054,A -85,B 0,C 180,E1 -20804.158,E2 -20804.158} C_VEL
LIN {X 0,Y 339.943,Z 245.947,A -85,B 0,C 180,E1 -20805.591,E2 -20805.591} C_VEL
LIN {X 0,Y 334.315,Z 241.909,A -85,B 0,C 180,E1 -20807.116,E2 -20807.116} C_VEL
LIN {X 0,Y 326.823,Z 236.779,A -85,B 0,C 180,E1 -20808.886,E2 -20808.886} C_VEL
LIN {X 0,Y 319.715,Z 231.508,A -85,B 0,C 180,E1 -20810.401,E2 -20810.401} C_VEL
LIN {X 0,Y 310.855,Z 225.076,A -85,B 0,C 180,E1 -20812.038,E2 -20812.038} C_VEL
LIN {X 0,Y 301.976,Z 218.197,A -85,B 0,C 180,E1 -20813.473,E2 -20813.473} C_VEL
LIN {X 0,Y 293.186,Z 211.137,A -85,B 0,C 180,E1 -20814.682,E2 -20814.682} C_VEL
LIN {X 0,Y 282.604,Z 202.144,A -85,B 0,C 180,E1 -20816.056,E2 -20816.056} C_VEL
LIN {X 0,Y 273.016,Z 193.289,A -85,B 0,C 180,E1 -20817.325,E2 -20817.325} C_VEL
LIN {X 0,Y 259.716,Z 179.264,A -85,B 0,C 180,E1 -20819.3,E2 -20819.3} C_VEL
LIN {X 0,Y 250.278,Z 167.434,A -85,B 0,C 180,E1 -20820.917,E2 -20820.917} C_VEL
LIN {X 0,Y 241.047,Z 153.175,A -85,B 0,C 180,E1 -20822.745,E2 -20822.745} C_VEL
LIN {X 0,Y 229.278,Z 130.087,A -85,B 0,C 180,E1 -20825.539,E2 -20825.539} C_VEL
LIN {X 0,Y 221.074,Z 115.603,A -85,B 0,C 180,E1 -20827.665,E2 -20827.665} C_VEL
LIN {X 0,Y 216.462,Z 108.372,A -85,B 0,C 180,E1 -20828.922,E2 -20828.922} C_VEL
LIN {X 0,Y 214.249,Z 105.123,A -85,B 0,C 180,E1 -20829.553,E2 -20829.553} C_VEL
LIN {X 0,Y 213.829,Z 103.768,A -85,B 0,C 180,E1 -20829.871,E2 -20829.871} C_VEL
LIN {X 0,Y 213.743,Z 103.361,A -85,B 0,C 180,E1 -20830.403,E2 -20830.403} C_VEL
LIN {X 0,Y 213.7,Z 103.307,A -85,B 0,C 180,E1 -20833.68,E2 -20833.68} C_VEL
LIN {X 0,Y 213.727,Z 103.361,A -85,B 0,C 180,E1 -20836.338,E2 -20836.338} C_VEL
LIN {X 0,Y 213.735,Z 103.355,A -85,B 0,C 180,E1 -20841.337,E2 -20841.337} C_VEL
LIN {X 0,Y 213.766,Z 103.331,A -85,B 0,C 180,E1 -20846.021,E2 -20846.021} C_VEL
LIN {X 0,Y 213.758,Z 103.344,A -85,B 0,C 180,E1 -20850.452,E2 -20850.452} C_VEL
LIN {X 0,Y 213.799,Z 103.333,A -85,B 0,C 180,E1 -20854.703,E2 -20854.703} C_VEL
LIN {X 0,Y 213.812,Z 103.328,A -85,B 0,C 180,E1 -20858.804,E2 -20858.804} C_VEL
LIN {X 0,Y 213.943,Z 103.306,A -85,B 0,C 180,E1 -20862.805,E2 -20862.805} C_VEL
LIN {X 0,Y 213.981,Z 103.324,A -85,B 0,C 180,E1 -20866.709,E2 -20866.709} C_VEL
LIN {X 0,Y 214.167,Z 103.26,A -85,B 0,C 180,E1 -20870.557,E2 -20870.557} C_VEL
LIN {X 0,Y 214.228,Z 103.273,A -85,B 0,C 180,E1 -20872.461,E2 -20872.461} C_VEL
LIN {X 0,Y 214.446,Z 103.235,A -85,B 0,C 180,E1 -20878.123,E2 -20878.123} C_VEL
LIN {X 0,Y 214.547,Z 103.21,A -85,B 0,C 180,E1 -20880.001,E2 -20880.001} C_VEL
LIN {X 0,Y 214.446,Z 103.238,A -85,B 0,C 180,E1 -20881.879,E2 -20881.879} C_VEL
LIN {X 0,Y 214.229,Z 103.269,A -85,B 0,C 180,E1 -20887.541,E2 -20887.541} C_VEL
LIN {X 0,Y 214.046,Z 103.284,A -85,B 0,C 180,E1 -20891.363,E2 -20891.363} C_VEL
LIN {X 0,Y 213.936,Z 103.329,A -85,B 0,C 180,E1 -20895.238,E2 -20895.238} C_VEL
LIN {X 0,Y 213.841,Z 103.302,A -85,B 0,C 180,E1 -20899.188,E2 -20899.188} C_VEL
LIN {X 0,Y 213.849,Z 103.346,A -85,B 0,C 180,E1 -20903.228,E2 -20903.228} C_VEL
LIN {X 0,Y 213.831,Z 103.313,A -85,B 0,C 180,E1 -20907.451,E2 -20907.451} C_VEL
LIN {X 0,Y 213.769,Z 103.352,A -85,B 0,C 180,E1 -20911.738,E2 -20911.738} C_VEL
LIN {X 0,Y 213.746,Z 103.348,A -85,B 0,C 180,E1 -20916.289,E2 -20916.289} C_VEL
LIN {X 0,Y 213.713,Z 103.348,A -85,B 0,C 180,E1 -20921.126,E2 -20921.126} C_VEL
LIN {X 0,Y 213.743,Z 103.496,A -85,B 0,C 180,E1 -20925.657,E2 -20925.657} C_VEL
LIN {X 0,Y 215.27,Z 109.884,A -85,B 0,C 180,E1 -20930.114,E2 -20930.114} C_VEL
LIN {X 0,Y 215.572,Z 110.882,A -85,B 0,C 180,E1 -20930.563,E2 -20930.563} C_VEL
LIN {X 0,Y 217.783,Z 114.99,A -85,B 0,C 180,E1 -20931.256,E2 -20931.256} C_VEL
LIN {X 0,Y 224.757,Z 129.028,A -85,B 0,C 180,E1 -20933.209,E2 -20933.209} C_VEL
LIN {X 0,Y 231.771,Z 145.022,A -85,B 0,C 180,E1 -20935.079,E2 -20935.079} C_VEL
LIN {X 0,Y 232.771,Z 148.79,A -85,B 0,C 180,E1 -20935.388,E2 -20935.388} C_VEL
LIN {X 0,Y 235.575,Z 165.515,A -85,B 0,C 180,E1 -20936.454,E2 -20936.454} C_VEL
LIN {X 0,Y 236.065,Z 169.522,A -85,B 0,C 180,E1 -20936.675,E2 -20936.675} C_VEL
LIN {X 0,Y 234.34,Z 212.004,A -85,B 0,C 180,E1 -20937.916,E2 -20937.916} C_VEL
LIN {X 0,Y 233.481,Z 217.828,A -85,B 0,C 180,E1 -20938.054,E2 -20938.054} C_VEL
LIN {X 0,Y 230.251,Z 227.215,A -85,B 0,C 180,E1 -20938.127,E2 -20938.127} C_VEL
LIN {X 0,Y 226.557,Z 236.391,A -85,B 0,C 180,E1 -20938.353,E2 -20938.353} C_VEL
LIN {X 0,Y 224.986,Z 241.883,A -85,B 0,C 180,E1 -20938.741,E2 -20938.741} C_VEL
LIN {X 0,Y 222.779,Z 253.209,A -85,B 0,C 180,E1 -20939.947,E2 -20939.947} C_VEL
LIN {X 0,Y 220.738,Z 262.482,A -85,B 0,C 180,E1 -20941.213,E2 -20941.213} C_VEL
LIN {X 0,Y 218.423,Z 271.422,A -85,B 0,C 180,E1 -20942.709,E2 -20942.709} C_VEL
LIN {X 0,Y 216.055,Z 279.948,A -85,B 0,C 180,E1 -20944.469,E2 -20944.469} C_VEL
LIN {X 0,Y 213.903,Z 287.164,A -85,B 0,C 180,E1 -20946.266,E2 -20946.266} C_VEL
LIN {X 0,Y 212.011,Z 293.503,A -85,B 0,C 180,E1 -20948.155,E2 -20948.155} C_VEL
LIN {X 0,Y 210.01,Z 299.903,A -85,B 0,C 180,E1 -20950.449,E2 -20950.449} C_VEL
LIN {X 0,Y 208.63,Z 304.406,A -85,B 0,C 180,E1 -20952.351,E2 -20952.351} C_VEL
LIN {X 0,Y 206.788,Z 309.896,A -85,B 0,C 180,E1 -20955.232,E2 -20955.232} C_VEL
LIN {X 0,Y 205.567,Z 314.224,A -85,B 0,C 180,E1 -20958.163,E2 -20958.163} C_VEL
LIN {X 0,Y 205.022,Z 316.595,A -85,B 0,C 180,E1 -20960.131,E2 -20960.131} C_VEL
LIN {X 0,Y 204.627,Z 318.398,A -85,B 0,C 180,E1 -20962.104,E2 -20962.104} C_VEL
LIN {X 0,Y 204.339,Z 320.853,A -85,B 0,C 180,E1 -20966.056,E2 -20966.056} C_VEL
LIN {X 0,Y 204.332,Z 321.446,A -85,B 0,C 180,E1 -20968.029,E2 -20968.029} C_VEL
LIN {X 0,Y 204.443,Z 321.604,A -85,B 0,C 180,E1 -20970,E2 -20970} C_VEL
LIN {X 0,Y 204.331,Z 321.446,A -85,B 0,C 180,E1 -20971.971,E2 -20971.971} C_VEL
LIN {X 0,Y 204.299,Z 320.852,A -85,B 0,C 180,E1 -20973.945,E2 -20973.945} C_VEL
LIN {X 0,Y 204.627,Z 318.398,A -85,B 0,C 180,E1 -20977.896,E2 -20977.896} C_VEL
LIN {X 0,Y 205.276,Z 315.443,A -85,B 0,C 180,E1 -20980.854,E2 -20980.854} C_VEL
LIN {X 0,Y 206.277,Z 311.449,A -85,B 0,C 180,E1 -20983.798,E2 -20983.798} C_VEL
LIN {X 0,Y 207.941,Z 306.321,A -85,B 0,C 180,E1 -20986.695,E2 -20986.695} C_VEL
LIN {X 0,Y 209.606,Z 301.058,A -85,B 0,C 180,E1 -20989.081,E2 -20989.081} C_VEL
LIN {X 0,Y 211.722,Z 294.745,A -85,B 0,C 180,E1 -20991.416,E2 -20991.416} C_VEL
LIN {X 0,Y 213.442,Z 288.792,A -85,B 0,C 180,E1 -20993.274,E2 -20993.274} C_VEL
LIN {X 0,Y 215.502,Z 281.866,A -85,B 0,C 180,E1 -20995.085,E2 -20995.085} C_VEL
LIN {X 0,Y 217.866,Z 273.692,A -85,B 0,C 180,E1 -20996.847,E2 -20996.847} C_VEL
LIN {X 0,Y 220.071,Z 265.184,A -85,B 0,C 180,E1 -20998.362,E2 -20998.362} C_VEL
LIN {X 0,Y 222.116,Z 256.473,A -85,B 0,C 180,E1 -20999.63,E2 -20999.63} C_VEL
LIN {X 0,Y 223.909,Z 247.725,A -85,B 0,C 180,E1 -21000.667,E2 -21000.667} C_VEL
LIN {X 0,Y 225.595,Z 237.927,A -85,B 0,C 180,E1 -21001.585,E2 -21001.585} C_VEL
LIN {X 0,Y 226.992,Z 227.83,A -85,B 0,C 180,E1 -21002.295,E2 -21002.295} C_VEL
LIN {X 0,Y 228.008,Z 217.013,A -85,B 0,C 180,E1 -21002.831,E2 -21002.831} C_VEL
LIN {X 0,Y 230.117,Z 170.352,A -85,B 0,C 180,E1 -21004.267,E2 -21004.267} C_VEL
LIN {X 0,Y 228.143,Z 157.163,A -85,B 0,C 180,E1 -21005.097,E2 -21005.097} C_VEL
LIN {X 0,Y 226.561,Z 148.723,A -85,B 0,C 180,E1 -21005.698,E2 -21005.698} C_VEL
LIN {X 0,Y 220.566,Z 134.691,A -85,B 0,C 180,E1 -21007.377,E2 -21007.377} C_VEL
LIN {X 0,Y 214.128,Z 121.555,A -85,B 0,C 180,E1 -21009.249,E2 -21009.249} C_VEL
LIN {X 0,Y 210.156,Z 114.327,A -85,B 0,C 180,E1 -21010.45,E2 -21010.45} C_VEL
LIN {X 0,Y 208.186,Z 110.418,A -85,B 0,C 180,E1 -21011.181,E2 -21011.181} C_VEL
LIN {X 0,Y 207.273,Z 106.889,A -85,B 0,C 180,E1 -21013.575,E2 -21013.575} C_VEL
LIN {X 0,Y 206.664,Z 104.243,A -85,B 0,C 180,E1 -21015.728,E2 -21015.728} C_VEL
LIN {X 0,Y 206.662,Z 104.222,A -85,B 0,C 180,E1 -21019.748,E2 -21019.748} C_VEL
LIN {X 0,Y 206.701,Z 104.212,A -85,B 0,C 180,E1 -21024.688,E2 -21024.688} C_VEL
LIN {X 0,Y 206.709,Z 104.237,A -85,B 0,C 180,E1 -21029.336,E2 -21029.336} C_VEL
LIN {X 0,Y 206.734,Z 104.198,A -85,B 0,C 180,E1 -21033.771,E2 -21033.771} C_VEL
LIN {X 0,Y 206.76,Z 104.219,A -85,B 0,C 180,E1 -21038.042,E2 -21038.042} C_VEL
LIN {X 0,Y 206.875,Z 104.172,A -85,B 0,C 180,E1 -21042.196,E2 -21042.196} C_VEL
LIN {X 0,Y 206.916,Z 104.205,A -85,B 0,C 180,E1 -21046.245,E2 -21046.245} C_VEL
LIN {X 0,Y 207.107,Z 104.136,A -85,B 0,C 180,E1 -21050.23,E2 -21050.23} C_VEL
LIN {X 0,Y 207.17,Z 104.143,A -85,B 0,C 180,E1 -21052.2,E2 -21052.2} C_VEL
LIN {X 0,Y 207.383,Z 104.118,A -85,B 0,C 180,E1 -21058.057,E2 -21058.057} C_VEL
LIN {X 0,Y 207.512,Z 104.085,A -85,B 0,C 180,E1 -21059.999,E2 -21059.999} C_VEL
LIN {X 0,Y 207.383,Z 104.115,A -85,B 0,C 180,E1 -21061.941,E2 -21061.941} C_VEL
LIN {X 0,Y 207.168,Z 104.146,A -85,B 0,C 180,E1 -21067.798,E2 -21067.798} C_VEL
LIN {X 0,Y 206.982,Z 104.168,A -85,B 0,C 180,E1 -21071.754,E2 -21071.754} C_VEL
LIN {X 0,Y 206.868,Z 104.21,A -85,B 0,C 180,E1 -21075.77,E2 -21075.77} C_VEL
LIN {X 0,Y 206.782,Z 104.187,A -85,B 0,C 180,E1 -21079.868,E2 -21079.868} C_VEL
LIN {X 0,Y 206.762,Z 104.228,A -85,B 0,C 180,E1 -21084.071,E2 -21084.071} C_VEL
LIN {X 0,Y 206.735,Z 104.203,A -85,B 0,C 180,E1 -21088.419,E2 -21088.419} C_VEL
LIN {X 0,Y 206.703,Z 104.218,A -85,B 0,C 180,E1 -21092.955,E2 -21092.955} C_VEL
LIN {X 0,Y 206.72,Z 104.21,A -85,B 0,C 180,E1 -21095.319,E2 -21095.319} C_VEL
LIN {X 0,Y 206.668,Z 104.22,A -85,B 0,C 180,E1 -21100.248,E2 -21100.248} C_VEL
LIN {X 0,Y 206.645,Z 104.222,A -85,B 0,C 180,E1 -21104.422,E2 -21104.422} C_VEL
LIN {X 0,Y 206.685,Z 104.418,A -85,B 0,C 180,E1 -21108.335,E2 -21108.335} C_VEL
LIN {X 0,Y 206.992,Z 105.58,A -85,B 0,C 180,E1 -21108.767,E2 -21108.767} C_VEL
LIN {X 0,Y 208.656,Z 108.294,A -85,B 0,C 180,E1 -21109.309,E2 -21109.309} C_VEL
LIN {X 0,Y 209.686,Z 109.632,A -85,B 0,C 180,E1 -21109.611,E2 -21109.611} C_VEL
LIN {X 0,Y 218.531,Z 123.671,A -85,B 0,C 180,E1 -21112.145,E2 -21112.145} C_VEL
LIN {X 0,Y 227.217,Z 139.779,A -85,B 0,C 180,E1 -21114.457,E2 -21114.457} C_VEL
LIN {X 0,Y 236.095,Z 157.549,A -85,B 0,C 180,E1 -21116.63,E2 -21116.63} C_VEL
LIN {X 0,Y 244.313,Z 170.447,A -85,B 0,C 180,E1 -21118.337,E2 -21118.337} C_VEL
LIN {X 0,Y 252.332,Z 180.968,A -85,B 0,C 180,E1 -21119.802,E2 -21119.802} C_VEL
LIN {X 0,Y 264.524,Z 194.547,A -85,B 0,C 180,E1 -21121.751,E2 -21121.751} C_VEL
LIN {X 0,Y 276.26,Z 205.847,A -85,B 0,C 180,E1 -21123.425,E2 -21123.425} C_VEL
LIN {X 0,Y 286.635,Z 214.904,A -85,B 0,C 180,E1 -21124.912,E2 -21124.912} C_VEL
LIN {X 0,Y 296.848,Z 223.203,A -85,B 0,C 180,E1 -21126.368,E2 -21126.368} C_VEL
LIN {X 0,Y 304.245,Z 228.93,A -85,B 0,C 180,E1 -21127.514,E2 -21127.514} C_VEL
LIN {X 0,Y 312.027,Z 234.642,A -85,B 0,C 180,E1 -21128.877,E2 -21128.877} C_VEL
LIN {X 0,Y 318.782,Z 239.715,A -85,B 0,C 180,E1 -21130.228,E2 -21130.228} C_VEL
LIN {X 0,Y 325.65,Z 244.491,A -85,B 0,C 180,E1 -21131.727,E2 -21131.727} C_VEL
LIN {X 0,Y 330.757,Z 248.061,A -85,B 0,C 180,E1 -21132.971,E2 -21132.971} C_VEL
LIN {X 0,Y 335.747,Z 251.727,A -85,B 0,C 180,E1 -21134.34,E2 -21134.34} C_VEL
LIN {X 0,Y 340.733,Z 254.903,A -85,B 0,C 180,E1 -21135.792,E2 -21135.792} C_VEL
LIN {X 0,Y 345.686,Z 257.752,A -85,B 0,C 180,E1 -21137.383,E2 -21137.383} C_VEL
LIN {X 0,Y 350.427,Z 261.283,A -85,B 0,C 180,E1 -21139.329,E2 -21139.329} C_VEL
LIN {X 0,Y 355.177,Z 264.281,A -85,B 0,C 180,E1 -21141.631,E2 -21141.631} C_VEL
LIN {X 0,Y 357.948,Z 265.727,A -85,B 0,C 180,E1 -21143.235,E2 -21143.235} C_VEL
LIN {X 0,Y 359.991,Z 266.594,A -85,B 0,C 180,E1 -21144.651,E2 -21144.651} C_VEL
LIN {X 0,Y 362.108,Z 267.339,A -85,B 0,C 180,E1 -21146.662,E2 -21146.662} C_VEL
LIN {X 0,Y 362.817,Z 267.672,A -85,B 0,C 180,E1 -21147.78,E2 -21147.78} C_VEL
LIN {X 0,Y 363.155,Z 267.985,A -85,B 0,C 180,E1 -21148.891,E2 -21148.891} C_VEL
LIN {X 0,Y 363.365,Z 267.945,A -85,B 0,C 180,E1 -21150,E2 -21150} C_VEL
LIN {X 0,Y 363.197,Z 267.911,A -85,B 0,C 180,E1 -21151.109,E2 -21151.109} C_VEL
LIN {X 0,Y 362.823,Z 267.639,A -85,B 0,C 180,E1 -21152.22,E2 -21152.22} C_VEL
LIN {X 0,Y 362.119,Z 267.288,A -85,B 0,C 180,E1 -21153.338,E2 -21153.338} C_VEL
LIN {X 0,Y 359.983,Z 266.604,A -85,B 0,C 180,E1 -21155.336,E2 -21155.336} C_VEL
LIN {X 0,Y 357.943,Z 265.704,A -85,B 0,C 180,E1 -21156.765,E2 -21156.765} C_VEL
LIN {X 0,Y 355.181,Z 264.309,A -85,B 0,C 180,E1 -21158.372,E2 -21158.372} C_VEL
LIN {X 0,Y 350.419,Z 261.285,A -85,B 0,C 180,E1 -21160.663,E2 -21160.663} C_VEL
LIN {X 0,Y 345.67,Z 257.772,A -85,B 0,C 180,E1 -21162.605,E2 -21162.605} C_VEL
LIN {X 0,Y 340.257,Z 254.594,A -85,B 0,C 180,E1 -21164.351,E2 -21164.351} C_VEL
LIN {X 0,Y 333.067,Z 249.815,A -85,B 0,C 180,E1 -21166.404,E2 -21166.404} C_VEL
LIN {X 0,Y 327.582,Z 245.756,A -85,B 0,C 180,E1 -21167.83,E2 -21167.83} C_VEL
LIN {X 0,Y 320.437,Z 240.922,A -85,B 0,C 180,E1 -21169.424,E2 -21169.424} C_VEL
LIN {X 0,Y 311.972,Z 234.631,A -85,B 0,C 180,E1 -21171.127,E2 -21171.127} C_VEL
LIN {X 0,Y 304.242,Z 228.919,A -85,B 0,C 180,E1 -21172.484,E2 -21172.484} C_VEL
LIN {X 0,Y 296.846,Z 223.196,A -85,B 0,C 180,E1 -21173.631,E2 -21173.631} C_VEL
LIN {X 0,Y 282.09,Z 211.126,A -85,B 0,C 180,E1 -21175.739,E2 -21175.739} C_VEL
LIN {X 0,Y 269.838,Z 199.874,A -85,B 0,C 180,E1 -21177.483,E2 -21177.483} C_VEL
LIN {X 0,Y 255.942,Z 185.266,A -85,B 0,C 180,E1 -21179.589,E2 -21179.589} C_VEL
LIN {X 0,Y 246.212,Z 173.184,A -85,B 0,C 180,E1 -21181.297,E2 -21181.297} C_VEL
LIN {X 0,Y 237.069,Z 159.222,A -85,B 0,C 180,E1 -21183.155,E2 -21183.155} C_VEL
LIN {X 0,Y 229.898,Z 145.347,A -85,B 0,C 180,E1 -21184.856,E2 -21184.856} C_VEL
LIN {X 0,Y 223.044,Z 131.806,A -85,B 0,C 180,E1 -21186.632,E2 -21186.632} C_VEL
LIN {X 0,Y 216.125,Z 119.773,A -85,B 0,C 180,E1 -21188.518,E2 -21188.518} C_VEL
LIN {X 0,Y 210.871,Z 111.634,A -85,B 0,C 180,E1 -21190.026,E2 -21190.026} C_VEL
LIN {X 0,Y 209.027,Z 108.649,A -85,B 0,C 180,E1 -21190.587,E2 -21190.587} C_VEL
LIN {X 0,Y 207.195,Z 106.074,A -85,B 0,C 180,E1 -21191.15,E2 -21191.15} C_VEL
LIN {X 0,Y 206.755,Z 104.764,A -85,B 0,C 180,E1 -21191.453,E2 -21191.453} C_VEL
LIN {X 0,Y 206.617,Z 104.221,A -85,B 0,C 180,E1 -21192.134,E2 -21192.134} C_VEL
LIN {X 0,Y 206.645,Z 104.222,A -85,B 0,C 180,E1 -21195.578,E2 -21195.578} C_VEL
LIN {X 0,Y 206.668,Z 104.22,A -85,B 0,C 180,E1 -21199.752,E2 -21199.752} C_VEL
LIN {X 0,Y 206.729,Z 104.209,A -85,B 0,C 180,E1 -21204.696,E2 -21204.696} C_VEL
LIN {X 0,Y 206.706,Z 104.237,A -85,B 0,C 180,E1 -21209.337,E2 -21209.337} C_VEL
LIN {X 0,Y 206.73,Z 104.202,A -85,B 0,C 180,E1 -21213.773,E2 -21213.773} C_VEL
LIN {X 0,Y 206.757,Z 104.219,A -85,B 0,C 180,E1 -21218.044,E2 -21218.044} C_VEL
LIN {X 0,Y 206.872,Z 104.178,A -85,B 0,C 180,E1 -21222.198,E2 -21222.198} C_VEL
LIN {X 0,Y 206.914,Z 104.208,A -85,B 0,C 180,E1 -21226.247,E2 -21226.247} C_VEL
LIN {X 0,Y 207.106,Z 104.138,A -85,B 0,C 180,E1 -21230.232,E2 -21230.232} C_VEL
LIN {X 0,Y 207.168,Z 104.146,A -85,B 0,C 180,E1 -21232.202,E2 -21232.202} C_VEL
LIN {X 0,Y 207.383,Z 104.115,A -85,B 0,C 180,E1 -21238.059,E2 -21238.059} C_VEL
LIN {X 0,Y 207.512,Z 104.085,A -85,B 0,C 180,E1 -21240.001,E2 -21240.001} C_VEL
LIN {X 0,Y 207.383,Z 104.118,A -85,B 0,C 180,E1 -21241.943,E2 -21241.943} C_VEL
LIN {X 0,Y 207.17,Z 104.143,A -85,B 0,C 180,E1 -21247.8,E2 -21247.8} C_VEL
LIN {X 0,Y 206.983,Z 104.168,A -85,B 0,C 180,E1 -21251.756,E2 -21251.756} C_VEL
LIN {X 0,Y 206.869,Z 104.203,A -85,B 0,C 180,E1 -21255.772,E2 -21255.772} C_VEL
LIN {X 0,Y 206.785,Z 104.184,A -85,B 0,C 180,E1 -21259.87,E2 -21259.87} C_VEL
LIN {X 0,Y 206.765,Z 104.222,A -85,B 0,C 180,E1 -21264.073,E2 -21264.073} C_VEL
LIN {X 0,Y 206.739,Z 104.203,A -85,B 0,C 180,E1 -21268.421,E2 -21268.421} C_VEL
LIN {X 0,Y 206.701,Z 104.214,A -85,B 0,C 180,E1 -21272.958,E2 -21272.958} C_VEL
LIN {X 0,Y 206.683,Z 104.24,A -85,B 0,C 180,E1 -21277.74,E2 -21277.74} C_VEL
LIN {X 0,Y 206.643,Z 104.232,A -85,B 0,C 180,E1 -21281.563,E2 -21281.563} C_VEL
LIN {X 0,Y 206.715,Z 104.447,A -85,B 0,C 180,E1 -21284.58,E2 -21284.58} C_VEL
LIN {X 0,Y 208.097,Z 110.204,A -85,B 0,C 180,E1 -21288.719,E2 -21288.719} C_VEL
LIN {X 0,Y 208.869,Z 112.179,A -85,B 0,C 180,E1 -21289.152,E2 -21289.152} C_VEL
LIN {X 0,Y 213.989,Z 121.152,A -85,B 0,C 180,E1 -21290.703,E2 -21290.703} C_VEL
LIN {X 0,Y 220.87,Z 135.204,A -85,B 0,C 180,E1 -21292.703,E2 -21292.703} C_VEL
LIN {X 0,Y 226.841,Z 149.6,A -85,B 0,C 180,E1 -21294.385,E2 -21294.385} C_VEL
LIN {X 0,Y 229.914,Z 168.323,A -85,B 0,C 180,E1 -21295.624,E2 -21295.624} C_VEL
LIN {X 0,Y 230.09,Z 171.008,A -85,B 0,C 180,E1 -21295.753,E2 -21295.753} C_VEL
LIN {X 0,Y 228.04,Z 217.098,A -85,B 0,C 180,E1 -21297.176,E2 -21297.176} C_VEL
LIN {X 0,Y 226.937,Z 228.553,A -85,B 0,C 180,E1 -21297.751,E2 -21297.751} C_VEL
LIN {X 0,Y 224.986,Z 241.883,A -85,B 0,C 180,E1 -21298.741,E2 -21298.741} C_VEL
LIN {X 0,Y 223.357,Z 247.381,A -85,B 0,C 180,E1 -21299.199,E2 -21299.199} C_VEL
LIN {X 0,Y 219.145,Z 255.966,A -85,B 0,C 180,E1 -21299.828,E2 -21299.828} C_VEL
LIN {X 0,Y 214.724,Z 264.25,A -85,B 0,C 180,E1 -21300.649,E2 -21300.649} C_VEL
LIN {X 0,Y 212.783,Z 269.044,A -85,B 0,C 180,E1 -21301.406,E2 -21301.406} C_VEL
LIN {X 0,Y 210.268,Z 277.839,A -85,B 0,C 180,E1 -21303.178,E2 -21303.178} C_VEL
LIN {X 0,Y 207.396,Z 286.973,A -85,B 0,C 180,E1 -21305.474,E2 -21305.474} C_VEL
LIN {X 0,Y 205.202,Z 293.933,A -85,B 0,C 180,E1 -21307.63,E2 -21307.63} C_VEL
LIN {X 0,Y 203.327,Z 299.713,A -85,B 0,C 180,E1 -21309.779,E2 -21309.779} C_VEL
LIN {X 0,Y 201.837,Z 304.215,A -85,B 0,C 180,E1 -21311.737,E2 -21311.737} C_VEL
LIN {X 0,Y 199.89,Z 309.704,A -85,B 0,C 180,E1 -21314.711,E2 -21314.711} C_VEL
LIN {X 0,Y 198.59,Z 314.033,A -85,B 0,C 180,E1 -21317.741,E2 -21317.741} C_VEL
LIN {X 0,Y 197.999,Z 316.404,A -85,B 0,C 180,E1 -21319.777,E2 -21319.777} C_VEL
LIN {X 0,Y 197.578,Z 318.207,A -85,B 0,C 180,E1 -21321.82,E2 -21321.82} C_VEL
LIN {X 0,Y 197.247,Z 320.713,A -85,B 0,C 180,E1 -21326.086,E2 -21326.086} C_VEL
LIN {X 0,Y 197.24,Z 321.256,A -85,B 0,C 180,E1 -21327.958,E2 -21327.958} C_VEL
LIN {X 0,Y 197.344,Z 321.414,A -85,B 0,C 180,E1 -21330,E2 -21330} C_VEL
LIN {X 0,Y 197.237,Z 321.256,A -85,B 0,C 180,E1 -21332.042,E2 -21332.042} C_VEL
LIN {X 0,Y 197.21,Z 320.662,A -85,B 0,C 180,E1 -21334.087,E2 -21334.087} C_VEL
LIN {X 0,Y 197.578,Z 318.207,A -85,B 0,C 180,E1 -21338.18,E2 -21338.18} C_VEL
LIN {X 0,Y 198.265,Z 315.252,A -85,B 0,C 180,E1 -21341.242,E2 -21341.242} C_VEL
LIN {X 0,Y 199.353,Z 311.258,A -85,B 0,C 180,E1 -21344.287,E2 -21344.287} C_VEL
LIN {X 0,Y 201.128,Z 306.13,A -85,B 0,C 180,E1 -21347.278,E2 -21347.278} C_VEL
LIN {X 0,Y 202.892,Z 300.867,A -85,B 0,C 180,E1 -21349.739,E2 -21349.739} C_VEL
LIN {X 0,Y 205.067,Z 294.553,A -85,B 0,C 180,E1 -21352.147,E2 -21352.147} C_VEL
LIN {X 0,Y 207.411,Z 286.973,A -85,B 0,C 180,E1 -21354.524,E2 -21354.524} C_VEL
LIN {X 0,Y 210.294,Z 277.84,A -85,B 0,C 180,E1 -21356.819,E2 -21356.819} C_VEL
LIN {X 0,Y 213.496,Z 266.344,A -85,B 0,C 180,E1 -21359.048,E2 -21359.048} C_VEL
LIN {X 0,Y 215.95,Z 256.281,A -85,B 0,C 180,E1 -21360.564,E2 -21360.564} C_VEL
LIN {X 0,Y 218.031,Z 246.528,A -85,B 0,C 180,E1 -21361.723,E2 -21361.723} C_VEL
LIN {X 0,Y 219.59,Z 237.737,A -85,B 0,C 180,E1 -21362.553,E2 -21362.553} C_VEL
LIN {X 0,Y 221.076,Z 227.175,A -85,B 0,C 180,E1 -21363.305,E2 -21363.305} C_VEL
LIN {X 0,Y 222.114,Z 216.568,A -85,B 0,C 180,E1 -21363.83,E2 -21363.83} C_VEL
LIN {X 0,Y 224.187,Z 170.37,A -85,B 0,C 180,E1 -21365.298,E2 -21365.298} C_VEL
LIN {X 0,Y 221.217,Z 151.971,A -85,B 0,C 180,E1 -21366.564,E2 -21366.564} C_VEL
LIN {X 0,Y 215.277,Z 137.885,A -85,B 0,C 180,E1 -21368.32,E2 -21368.32} C_VEL
LIN {X 0,Y 208.504,Z 123.904,A -85,B 0,C 180,E1 -21370.411,E2 -21370.411} C_VEL
LIN {X 0,Y 202.96,Z 114.226,A -85,B 0,C 180,E1 -21372.198,E2 -21372.198} C_VEL
LIN {X 0,Y 200.843,Z 110.268,A -85,B 0,C 180,E1 -21373.016,E2 -21373.016} C_VEL
LIN {X 0,Y 200.323,Z 107.922,A -85,B 0,C 180,E1 -21374.561,E2 -21374.561} C_VEL
LIN {X 0,Y 199.603,Z 105.159,A -85,B 0,C 180,E1 -21376.889,E2 -21376.889} C_VEL
LIN {X 0,Y 199.612,Z 105.103,A -85,B 0,C 180,E1 -21380.767,E2 -21380.767} C_VEL
LIN {X 0,Y 199.613,Z 105.09,A -85,B 0,C 180,E1 -21385.712,E2 -21385.712} C_VEL
LIN {X 0,Y 199.695,Z 105.101,A -85,B 0,C 180,E1 -21388.135,E2 -21388.135} C_VEL
LIN {X 0,Y 199.687,Z 105.073,A -85,B 0,C 180,E1 -21392.771,E2 -21392.771} C_VEL
LIN {X 0,Y 199.74,Z 105.102,A -85,B 0,C 180,E1 -21397.228,E2 -21397.228} C_VEL
LIN {X 0,Y 199.798,Z 105.05,A -85,B 0,C 180,E1 -21401.757,E2 -21401.757} C_VEL
LIN {X 0,Y 199.85,Z 105.088,A -85,B 0,C 180,E1 -21405.748,E2 -21405.748} C_VEL
LIN {X 0,Y 200.071,Z 105.012,A -85,B 0,C 180,E1 -21409.883,E2 -21409.883} C_VEL
LIN {X 0,Y 200.037,Z 105.061,A -85,B 0,C 180,E1 -21413.949,E2 -21413.949} C_VEL
LIN {X 0,Y 200.323,Z 104.997,A -85,B 0,C 180,E1 -21417.988,E2 -21417.988} C_VEL
LIN {X 0,Y 200.477,Z 104.961,A -85,B 0,C 180,E1 -21419.999,E2 -21419.999} C_VEL
LIN {X 0,Y 200.032,Z 105.063,A -85,B 0,C 180,E1 -21424.028,E2 -21424.028} C_VEL
LIN {X 0,Y 200.112,Z 105.02,A -85,B 0,C 180,E1 -21428.075,E2 -21428.075} C_VEL
LIN {X 0,Y 199.914,Z 105.054,A -85,B 0,C 180,E1 -21432.176,E2 -21432.176} C_VEL
LIN {X 0,Y 199.805,Z 105.078,A -85,B 0,C 180,E1 -21436.342,E2 -21436.342} C_VEL
LIN {X 0,Y 199.699,Z 105.075,A -85,B 0,C 180,E1 -21440.604,E2 -21440.604} C_VEL
LIN {X 0,Y 199.671,Z 105.096,A -85,B 0,C 180,E1 -21444.983,E2 -21444.983} C_VEL
LIN {X 0,Y 199.663,Z 105.097,A -85,B 0,C 180,E1 -21449.523,E2 -21449.523} C_VEL
LIN {X 0,Y 199.656,Z 105.103,A -85,B 0,C 180,E1 -21452.348,E2 -21452.348} C_VEL
LIN {X 0,Y 199.638,Z 105.108,A -85,B 0,C 180,E1 -21456.758,E2 -21456.758} C_VEL
LIN {X 0,Y 199.637,Z 105.101,A -85,B 0,C 180,E1 -21459.32,E2 -21459.32} C_VEL
LIN {X 0,Y 199.587,Z 105.111,A -85,B 0,C 180,E1 -21462.314,E2 -21462.314} C_VEL
LIN {X 0,Y 199.613,Z 105.233,A -85,B 0,C 180,E1 -21466.433,E2 -21466.433} C_VEL
LIN {X 0,Y 199.828,Z 106.246,A -85,B 0,C 180,E1 -21466.943,E2 -21466.943} C_VEL
LIN {X 0,Y 201.424,Z 109.046,A -85,B 0,C 180,E1 -21467.539,E2 -21467.539} C_VEL
LIN {X 0,Y 202.671,Z 110.447,A -85,B 0,C 180,E1 -21467.929,E2 -21467.929} C_VEL
LIN {X 0,Y 205.021,Z 113.96,A -85,B 0,C 180,E1 -21468.684,E2 -21468.684} C_VEL
LIN {X 0,Y 213.911,Z 128.207,A -85,B 0,C 180,E1 -21471.362,E2 -21471.362} C_VEL
LIN {X 0,Y 222.404,Z 144.177,A -85,B 0,C 180,E1 -21473.733,E2 -21473.733} C_VEL
LIN {X 0,Y 231.149,Z 161.878,A -85,B 0,C 180,E1 -21475.972,E2 -21475.972} C_VEL
LIN {X 0,Y 239.593,Z 175.239,A -85,B 0,C 180,E1 -21477.8,E2 -21477.8} C_VEL
LIN {X 0,Y 247.764,Z 186.028,A -85,B 0,C 180,E1 -21479.349,E2 -21479.349} C_VEL
LIN {X 0,Y 259.98,Z 199.731,A -85,B 0,C 180,E1 -21481.367,E2 -21481.367} C_VEL
LIN {X 0,Y 271.319,Z 210.854,A -85,B 0,C 180,E1 -21483.128,E2 -21483.128} C_VEL
LIN {X 0,Y 282.396,Z 220.582,A -85,B 0,C 180,E1 -21484.858,E2 -21484.858} C_VEL
LIN {X 0,Y 293.927,Z 229.876,A -85,B 0,C 180,E1 -21486.633,E2 -21486.633} C_VEL
LIN {X 0,Y 301.605,Z 235.832,A -85,B 0,C 180,E1 -21487.856,E2 -21487.856} C_VEL
LIN {X 0,Y 308.498,Z 240.796,A -85,B 0,C 180,E1 -21489.07,E2 -21489.07} C_VEL
LIN {X 0,Y 316.46,Z 246.812,A -85,B 0,C 180,E1 -21490.704,E2 -21490.704} C_VEL
LIN {X 0,Y 324.302,Z 252.112,A -85,B 0,C 180,E1 -21492.462,E2 -21492.462} C_VEL
LIN {X 0,Y 329.816,Z 256.19,A -85,B 0,C 180,E1 -21493.918,E2 -21493.918} C_VEL
LIN {X 0,Y 335.102,Z 259.697,A -85,B 0,C 180,E1 -21495.424,E2 -21495.424} C_VEL
LIN {X 0,Y 341.103,Z 263.203,A -85,B 0,C 180,E1 -21497.309,E2 -21497.309} C_VEL
LIN {X 0,Y 344.201,Z 265.513,A -85,B 0,C 180,E1 -21498.541,E2 -21498.541} C_VEL
LIN {X 0,Y 346.367,Z 267.096,A -85,B 0,C 180,E1 -21499.478,E2 -21499.478} C_VEL
LIN {X 0,Y 349.042,Z 268.865,A -85,B 0,C 180,E1 -21500.73,E2 -21500.73} C_VEL
LIN {X 0,Y 351.423,Z 270.208,A -85,B 0,C 180,E1 -21501.953,E2 -21501.953} C_VEL
LIN {X 0,Y 353.786,Z 271.431,A -85,B 0,C 180,E1 -21503.335,E2 -21503.335} C_VEL
LIN {X 0,Y 355.253,Z 272.066,A -85,B 0,C 180,E1 -21504.323,E2 -21504.323} C_VEL
LIN {X 0,Y 356.664,Z 272.68,A -85,B 0,C 180,E1 -21505.479,E2 -21505.479} C_VEL
LIN {X 0,Y 357.809,Z 273.027,A -85,B 0,C 180,E1 -21506.622,E2 -21506.622} C_VEL
LIN {X 0,Y 358.652,Z 273.435,A -85,B 0,C 180,E1 -21507.954,E2 -21507.954} C_VEL
LIN {X 0,Y 359.106,Z 273.629,A -85,B 0,C 180,E1 -21510,E2 -21510} C_VEL
LIN {X 0,Y 358.653,Z 273.374,A -85,B 0,C 180,E1 -21512.05,E2 -21512.05} C_VEL
LIN {X 0,Y 357.828,Z 272.967,A -85,B 0,C 180,E1 -21513.378,E2 -21513.378} C_VEL
LIN {X 0,Y 356.654,Z 272.649,A -85,B 0,C 180,E1 -21514.521,E2 -21514.521} C_VEL
LIN {X 0,Y 353.782,Z 271.412,A -85,B 0,C 180,E1 -21516.659,E2 -21516.659} C_VEL
LIN {X 0,Y 351.381,Z 270.229,A -85,B 0,C 180,E1 -21518.048,E2 -21518.048} C_VEL
LIN {X 0,Y 348.961,Z 268.791,A -85,B 0,C 180,E1 -21519.307,E2 -21519.307} C_VEL
LIN {X 0,Y 346.37,Z 267.064,A -85,B 0,C 180,E1 -21520.522,E2 -21520.522} C_VEL
LIN {X 0,Y 343.287,Z 264.908,A -85,B 0,C 180,E1 -21521.813,E2 -21521.813} C_VEL
LIN {X 0,Y 339.371,Z 262.21,A -85,B 0,C 180,E1 -21523.269,E2 -21523.269} C_VEL
LIN {X 0,Y 334.362,Z 259.205,A -85,B 0,C 180,E1 -21524.79,E2 -21524.79} C_VEL
LIN {X 0,Y 327.957,Z 254.826,A -85,B 0,C 180,E1 -21526.587,E2 -21526.587} C_VEL
LIN {X 0,Y 321.715,Z 250.396,A -85,B 0,C 180,E1 -21528.145,E2 -21528.145} C_VEL
LIN {X 0,Y 313.824,Z 244.9,A -85,B 0,C 180,E1 -21529.853,E2 -21529.853} C_VEL
LIN {X 0,Y 308.486,Z 240.812,A -85,B 0,C 180,E1 -21530.924,E2 -21530.924} C_VEL
LIN {X 0,Y 300.202,Z 234.74,A -85,B 0,C 180,E1 -21532.374,E2 -21532.374} C_VEL
LIN {X 0,Y 288.805,Z 225.958,A -85,B 0,C 180,E1 -21534.142,E2 -21534.142} C_VEL
LIN {X 0,Y 275.237,Z 214.455,A -85,B 0,C 180,E1 -21536.249,E2 -21536.249} C_VEL
LIN {X 0,Y 264.854,Z 204.632,A -85,B 0,C 180,E1 -21537.878,E2 -21537.878} C_VEL
LIN {X 0,Y 252.59,Z 191.732,A -85,B 0,C 180,E1 -21539.816,E2 -21539.816} C_VEL
LIN {X 0,Y 241.741,Z 178.348,A -85,B 0,C 180,E1 -21541.771,E2 -21541.771} C_VEL
LIN {X 0,Y 233.436,Z 165.689,A -85,B 0,C 180,E1 -21543.509,E2 -21543.509} C_VEL
LIN {X 0,Y 226.408,Z 152.724,A -85,B 0,C 180,E1 -21545.196,E2 -21545.196} C_VEL
LIN {X 0,Y 219.364,Z 138.223,A -85,B 0,C 180,E1 -21547.096,E2 -21547.096} C_VEL
LIN {X 0,Y 211.981,Z 124.961,A -85,B 0,C 180,E1 -21549.198,E2 -21549.198} C_VEL
LIN {X 0,Y 204.735,Z 113.646,A -85,B 0,C 180,E1 -21551.401,E2 -21551.401} C_VEL
LIN {X 0,Y 201.942,Z 109.556,A -85,B 0,C 180,E1 -21552.301,E2 -21552.301} C_VEL
LIN {X 0,Y 200.136,Z 107.051,A -85,B 0,C 180,E1 -21552.903,E2 -21552.903} C_VEL
LIN {X 0,Y 199.678,Z 105.621,A -85,B 0,C 180,E1 -21553.258,E2 -21553.258} C_VEL
LIN {X 0,Y 199.594,Z 105.195,A -85,B 0,C 180,E1 -21553.643,E2 -21553.643} C_VEL
LIN {X 0,Y 199.591,Z 105.107,A -85,B 0,C 180,E1 -21558.009,E2 -21558.009} C_VEL
LIN {X 0,Y 199.639,Z 105.101,A -85,B 0,C 180,E1 -21560.757,E2 -21560.757} C_VEL
LIN {X 0,Y 199.63,Z 105.09,A -85,B 0,C 180,E1 -21565.718,E2 -21565.718} C_VEL
LIN {X 0,Y 199.694,Z 105.106,A -85,B 0,C 180,E1 -21568.137,E2 -21568.137} C_VEL
LIN {X 0,Y 199.683,Z 105.075,A -85,B 0,C 180,E1 -21572.773,E2 -21572.773} C_VEL
LIN {X 0,Y 199.737,Z 105.104,A -85,B 0,C 180,E1 -21577.23,E2 -21577.23} C_VEL
LIN {X 0,Y 199.796,Z 105.055,A -85,B 0,C 180,E1 -21581.759,E2 -21581.759} C_VEL
LIN {X 0,Y 199.848,Z 105.092,A -85,B 0,C 180,E1 -21585.75,E2 -21585.75} C_VEL
LIN {X 0,Y 200.07,Z 105.014,A -85,B 0,C 180,E1 -21589.885,E2 -21589.885} C_VEL
LIN {X 0,Y 200.035,Z 105.063,A -85,B 0,C 180,E1 -21593.951,E2 -21593.951} C_VEL
LIN {X 0,Y 200.322,Z 104.994,A -85,B 0,C 180,E1 -21597.991,E2 -21597.991} C_VEL
LIN {X 0,Y 200.477,Z 104.961,A -85,B 0,C 180,E1 -21600.001,E2 -21600.001} C_VEL
LIN {X 0,Y 200.033,Z 105.065,A -85,B 0,C 180,E1 -21604.03,E2 -21604.03} C_VEL
LIN {X 0,Y 200.113,Z 105.017,A -85,B 0,C 180,E1 -21608.077,E2 -21608.077} C_VEL
LIN {X 0,Y 199.915,Z 105.054,A -85,B 0,C 180,E1 -21612.178,E2 -21612.178} C_VEL
LIN {X 0,Y 199.807,Z 105.071,A -85,B 0,C 180,E1 -21616.344,E2 -21616.344} C_VEL
LIN {X 0,Y 199.702,Z 105.074,A -85,B 0,C 180,E1 -21620.606,E2 -21620.606} C_VEL
LIN {X 0,Y 199.674,Z 105.09,A -85,B 0,C 180,E1 -21624.985,E2 -21624.985} C_VEL
LIN {X 0,Y 199.667,Z 105.099,A -85,B 0,C 180,E1 -21629.525,E2 -21629.525} C_VEL
LIN {X 0,Y 199.673,Z 105.096,A -85,B 0,C 180,E1 -21632.356,E2 -21632.356} C_VEL
LIN {X 0,Y 199.626,Z 105.113,A -85,B 0,C 180,E1 -21636.764,E2 -21636.764} C_VEL
LIN {X 0,Y 199.61,Z 105.102,A -85,B 0,C 180,E1 -21639.329,E2 -21639.329} C_VEL
LIN {X 0,Y 199.624,Z 105.271,A -85,B 0,C 180,E1 -21643.269,E2 -21643.269} C_VEL
LIN {X 0,Y 200.693,Z 109.693,A -85,B 0,C 180,E1 -21646.72,E2 -21646.72} C_VEL
LIN {X 0,Y 201.008,Z 110.697,A -85,B 0,C 180,E1 -21647.089,E2 -21647.089} C_VEL
LIN {X 0,Y 203.276,Z 114.667,A -85,B 0,C 180,E1 -21647.903,E2 -21647.903} C_VEL
LIN {X 0,Y 209.457,Z 125.734,A -85,B 0,C 180,E1 -21649.889,E2 -21649.889} C_VEL
LIN {X 0,Y 216.609,Z 140.826,A -85,B 0,C 180,E1 -21652.077,E2 -21652.077} C_VEL
LIN {X 0,Y 221.356,Z 152.487,A -85,B 0,C 180,E1 -21653.483,E2 -21653.483} C_VEL
LIN {X 0,Y 224.188,Z 170.352,A -85,B 0,C 180,E1 -21654.702,E2 -21654.702} C_VEL
LIN {X 0,Y 222.136,Z 216.637,A -85,B 0,C 180,E1 -21656.173,E2 -21656.173} C_VEL
LIN {X 0,Y 221.032,Z 227.865,A -85,B 0,C 180,E1 -21656.741,E2 -21656.741} C_VEL
LIN {X 0,Y 219.18,Z 240.309,A -85,B 0,C 180,E1 -21657.651,E2 -21657.651} C_VEL
LIN {X 0,Y 216.67,Z 253.019,A -85,B 0,C 180,E1 -21659.007,E2 -21659.007} C_VEL
LIN {X 0,Y 214.541,Z 262.292,A -85,B 0,C 180,E1 -21660.299,E2 -21660.299} C_VEL
LIN {X 0,Y 212.783,Z 269.044,A -85,B 0,C 180,E1 -21661.406,E2 -21661.406} C_VEL
LIN {X 0,Y 210.777,Z 273.791,A -85,B 0,C 180,E1 -21662.237,E2 -21662.237} C_VEL
LIN {X 0,Y 205.953,Z 281.105,A -85,B 0,C 180,E1 -21663.502,E2 -21663.502} C_VEL
LIN {X 0,Y 201.18,Z 287.968,A -85,B 0,C 180,E1 -21664.985,E2 -21664.985} C_VEL
LIN {X 0,Y 199.282,Z 291.779,A -85,B 0,C 180,E1 -21666.146,E2 -21666.146} C_VEL
LIN {X 0,Y 196.677,Z 299.522,A -85,B 0,C 180,E1 -21669.063,E2 -21669.063} C_VEL
LIN {X 0,Y 195.067,Z 304.023,A -85,B 0,C 180,E1 -21671.079,E2 -21671.079} C_VEL
LIN {X 0,Y 193.023,Z 309.513,A -85,B 0,C 180,E1 -21674.153,E2 -21674.153} C_VEL
LIN {X 0,Y 191.634,Z 313.842,A -85,B 0,C 180,E1 -21677.288,E2 -21677.288} C_VEL
LIN {X 0,Y 190.993,Z 316.213,A -85,B 0,C 180,E1 -21679.398,E2 -21679.398} C_VEL
LIN {X 0,Y 190.528,Z 318.016,A -85,B 0,C 180,E1 -21681.515,E2 -21681.515} C_VEL
LIN {X 0,Y 190.166,Z 320.472,A -85,B 0,C 180,E1 -21685.761,E2 -21685.761} C_VEL
LIN {X 0,Y 190.151,Z 321.065,A -85,B 0,C 180,E1 -21687.882,E2 -21687.882} C_VEL
LIN {X 0,Y 190.248,Z 321.224,A -85,B 0,C 180,E1 -21690,E2 -21690} C_VEL
LIN {X 0,Y 190.12,Z 320.67,A -85,B 0,C 180,E1 -21693.529,E2 -21693.529} C_VEL
LIN {X 0,Y 190.278,Z 319.409,A -85,B 0,C 180,E1 -21696.362,E2 -21696.362} C_VEL
LIN {X 0,Y 190.528,Z 318.016,A -85,B 0,C 180,E1 -21698.485,E2 -21698.485} C_VEL
LIN {X 0,Y 191.276,Z 315.06,A -85,B 0,C 180,E1 -21701.659,E2 -21701.659} C_VEL
LIN {X 0,Y 192.444,Z 311.066,A -85,B 0,C 180,E1 -21704.811,E2 -21704.811} C_VEL
LIN {X 0,Y 194.338,Z 305.938,A -85,B 0,C 180,E1 -21707.902,E2 -21707.902} C_VEL
LIN {X 0,Y 196.215,Z 300.676,A -85,B 0,C 180,E1 -21710.44,E2 -21710.44} C_VEL
LIN {X 0,Y 198.132,Z 295.419,A -85,B 0,C 180,E1 -21712.543,E2 -21712.543} C_VEL
LIN {X 0,Y 200.42,Z 288.409,A -85,B 0,C 180,E1 -21714.885,E2 -21714.885} C_VEL
LIN {X 0,Y 202.702,Z 281.484,A -85,B 0,C 180,E1 -21716.79,E2 -21716.79} C_VEL
LIN {X 0,Y 205.258,Z 273.31,A -85,B 0,C 180,E1 -21718.643,E2 -21718.643} C_VEL
LIN {X 0,Y 207.678,Z 264.803,A -85,B 0,C 180,E1 -21720.224,E2 -21720.224} C_VEL
LIN {X 0,Y 209.862,Z 256.091,A -85,B 0,C 180,E1 -21721.551,E2 -21721.551} C_VEL
LIN {X 0,Y 212.014,Z 246.337,A -85,B 0,C 180,E1 -21722.734,E2 -21722.734} C_VEL
LIN {X 0,Y 213.639,Z 237.546,A -85,B 0,C 180,E1 -21723.578,E2 -21723.578} C_VEL
LIN {X 0,Y 215.14,Z 227.224,A -85,B 0,C 180,E1 -21724.331,E2 -21724.331} C_VEL
LIN {X 0,Y 216.194,Z 217.176,A -85,B 0,C 180,E1 -21724.846,E2 -21724.846} C_VEL
LIN {X 0,Y 217.844,Z 184.686,A -85,B 0,C 180,E1 -21725.908,E2 -21725.908} C_VEL
LIN {X 0,Y 218.325,Z 171.09,A -85,B 0,C 180,E1 -21726.358,E2 -21726.358} C_VEL
LIN {X 0,Y 215.72,Z 154.641,A -85,B 0,C 180,E1 -21727.537,E2 -21727.537} C_VEL
LIN {X 0,Y 210.196,Z 141.439,A -85,B 0,C 180,E1 -21729.262,E2 -21729.262} C_VEL
LIN {X 0,Y 203.78,Z 128.087,A -85,B 0,C 180,E1 -21731.352,E2 -21731.352} C_VEL
LIN {X 0,Y 198.447,Z 118.645,A -85,B 0,C 180,E1 -21733.168,E2 -21733.168} C_VEL
LIN {X 0,Y 195.644,Z 113.934,A -85,B 0,C 180,E1 -21734.173,E2 -21734.173} C_VEL
LIN {X 0,Y 193.545,Z 109.898,A -85,B 0,C 180,E1 -21735.103,E2 -21735.103} C_VEL
LIN {X 0,Y 192.57,Z 106.144,A -85,B 0,C 180,E1 -21738.09,E2 -21738.09} C_VEL
LIN {X 0,Y 192.589,Z 105.985,A -85,B 0,C 180,E1 -21743.401,E2 -21743.401} C_VEL
LIN {X 0,Y 192.61,Z 105.968,A -85,B 0,C 180,E1 -21747.059,E2 -21747.059} C_VEL
LIN {X 0,Y 192.662,Z 105.953,A -85,B 0,C 180,E1 -21751.69,E2 -21751.69} C_VEL
LIN {X 0,Y 192.708,Z 105.976,A -85,B 0,C 180,E1 -21756.348,E2 -21756.348} C_VEL
LIN {X 0,Y 192.733,Z 105.929,A -85,B 0,C 180,E1 -21761.457,E2 -21761.457} C_VEL
LIN {X 0,Y 192.774,Z 105.969,A -85,B 0,C 180,E1 -21765.213,E2 -21765.213} C_VEL
LIN {X 0,Y 192.982,Z 105.896,A -85,B 0,C 180,E1 -21769.507,E2 -21769.507} C_VEL
LIN {X 0,Y 193.064,Z 105.89,A -85,B 0,C 180,E1 -21771.626,E2 -21771.626} C_VEL
LIN {X 0,Y 193.265,Z 105.875,A -85,B 0,C 180,E1 -21777.915,E2 -21777.915} C_VEL
LIN {X 0,Y 193.441,Z 105.836,A -85,B 0,C 180,E1 -21779.999,E2 -21779.999} C_VEL
LIN {X 0,Y 192.978,Z 105.943,A -85,B 0,C 180,E1 -21784.176,E2 -21784.176} C_VEL
LIN {X 0,Y 193.062,Z 105.893,A -85,B 0,C 180,E1 -21788.372,E2 -21788.372} C_VEL
LIN {X 0,Y 192.853,Z 105.94,A -85,B 0,C 180,E1 -21792.629,E2 -21792.629} C_VEL
LIN {X 0,Y 192.757,Z 105.944,A -85,B 0,C 180,E1 -21796.957,E2 -21796.957} C_VEL
LIN {X 0,Y 192.635,Z 105.965,A -85,B 0,C 180,E1 -21801.396,E2 -21801.396} C_VEL
LIN {X 0,Y 192.663,Z 105.98,A -85,B 0,C 180,E1 -21804.224,E2 -21804.224} C_VEL
LIN {X 0,Y 192.643,Z 105.961,A -85,B 0,C 180,E1 -21808.888,E2 -21808.888} C_VEL
LIN {X 0,Y 192.596,Z 105.971,A -85,B 0,C 180,E1 -21813.185,E2 -21813.185} C_VEL
LIN {X 0,Y 192.608,Z 105.981,A -85,B 0,C 180,E1 -21816.607,E2 -21816.607} C_VEL
LIN {X 0,Y 192.528,Z 105.98,A -85,B 0,C 180,E1 -21821.075,E2 -21821.075} C_VEL
LIN {X 0,Y 192.571,Z 106.205,A -85,B 0,C 180,E1 -21824.583,E2 -21824.583} C_VEL
LIN {X 0,Y 192.816,Z 107.228,A -85,B 0,C 180,E1 -21825.012,E2 -21825.012} C_VEL
LIN {X 0,Y 194.497,Z 110.06,A -85,B 0,C 180,E1 -21825.681,E2 -21825.681} C_VEL
LIN {X 0,Y 195.872,Z 111.653,A -85,B 0,C 180,E1 -21826.155,E2 -21826.155} C_VEL
LIN {X 0,Y 197.951,Z 114.808,A -85,B 0,C 180,E1 -21826.888,E2 -21826.888} C_VEL
LIN {X 0,Y 203.577,Z 123.239,A -85,B 0,C 180,E1 -21828.752,E2 -21828.752} C_VEL
LIN {X 0,Y 210.532,Z 134.883,A -85,B 0,C 180,E1 -21830.907,E2 -21830.907} C_VEL
LIN {X 0,Y 218.131,Z 149.706,A -85,B 0,C 180,E1 -21833.123,E2 -21833.123} C_VEL
LIN {X 0,Y 226.323,Z 166.348,A -85,B 0,C 180,E1 -21835.307,E2 -21835.307} C_VEL
LIN {X 0,Y 234.802,Z 179.885,A -85,B 0,C 180,E1 -21837.222,E2 -21837.222} C_VEL
LIN {X 0,Y 243.071,Z 190.92,A -85,B 0,C 180,E1 -21838.852,E2 -21838.852} C_VEL
LIN {X 0,Y 255.016,Z 204.51,A -85,B 0,C 180,E1 -21840.941,E2 -21840.941} C_VEL
LIN {X 0,Y 265.93,Z 215.498,A -85,B 0,C 180,E1 -21842.805,E2 -21842.805} C_VEL
LIN {X 0,Y 277.678,Z 225.932,A -85,B 0,C 180,E1 -21844.797,E2 -21844.797} C_VEL
LIN {X 0,Y 290.363,Z 236.02,A -85,B 0,C 180,E1 -21846.889,E2 -21846.889} C_VEL
LIN {X 0,Y 300.165,Z 243.588,A -85,B 0,C 180,E1 -21848.542,E2 -21848.542} C_VEL
LIN {X 0,Y 307.03,Z 248.491,A -85,B 0,C 180,E1 -21849.799,E2 -21849.799} C_VEL
LIN {X 0,Y 314.992,Z 254.333,A -85,B 0,C 180,E1 -21851.485,E2 -21851.485} C_VEL
LIN {X 0,Y 321.402,Z 258.751,A -85,B 0,C 180,E1 -21852.995,E2 -21852.995} C_VEL
LIN {X 0,Y 327.805,Z 263.334,A -85,B 0,C 180,E1 -21854.745,E2 -21854.745} C_VEL
LIN {X 0,Y 334.114,Z 267.192,A -85,B 0,C 180,E1 -21856.622,E2 -21856.622} C_VEL
LIN {X 0,Y 338.056,Z 269.782,A -85,B 0,C 180,E1 -21858.001,E2 -21858.001} C_VEL
LIN {X 0,Y 342.598,Z 273.045,A -85,B 0,C 180,E1 -21859.949,E2 -21859.949} C_VEL
LIN {X 0,Y 347.426,Z 275.916,A -85,B 0,C 180,E1 -21862.391,E2 -21862.391} C_VEL
LIN {X 0,Y 350.391,Z 277.313,A -85,B 0,C 180,E1 -21864.244,E2 -21864.244} C_VEL
LIN {X 0,Y 352.319,Z 278.135,A -85,B 0,C 180,E1 -21865.849,E2 -21865.849} C_VEL
LIN {X 0,Y 353.87,Z 278.694,A -85,B 0,C 180,E1 -21867.724,E2 -21867.724} C_VEL
LIN {X 0,Y 354.245,Z 278.987,A -85,B 0,C 180,E1 -21868.863,E2 -21868.863} C_VEL
LIN {X 0,Y 354.468,Z 278.973,A -85,B 0,C 180,E1 -21870,E2 -21870} C_VEL
LIN {X 0,Y 354.29,Z 278.925,A -85,B 0,C 180,E1 -21871.137,E2 -21871.137} C_VEL
LIN {X 0,Y 353.874,Z 278.664,A -85,B 0,C 180,E1 -21872.276,E2 -21872.276} C_VEL
LIN {X 0,Y 352.334,Z 278.113,A -85,B 0,C 180,E1 -21874.184,E2 -21874.184} C_VEL
LIN {X 0,Y 350.351,Z 277.309,A -85,B 0,C 180,E1 -21875.756,E2 -21875.756} C_VEL
LIN {X 0,Y 347.428,Z 275.952,A -85,B 0,C 180,E1 -21877.611,E2 -21877.611} C_VEL
LIN {X 0,Y 342.605,Z 273.012,A -85,B 0,C 180,E1 -21880.058,E2 -21880.058} C_VEL
LIN {X 0,Y 338.003,Z 269.764,A -85,B 0,C 180,E1 -21882.001,E2 -21882.001} C_VEL
LIN {X 0,Y 334.124,Z 267.208,A -85,B 0,C 180,E1 -21883.378,E2 -21883.378} C_VEL
LIN {X 0,Y 327.807,Z 263.316,A -85,B 0,C 180,E1 -21885.256,E2 -21885.256} C_VEL
LIN {X 0,Y 321.394,Z 258.719,A -85,B 0,C 180,E1 -21887.006,E2 -21887.006} C_VEL
LIN {X 0,Y 314.985,Z 254.335,A -85,B 0,C 180,E1 -21888.511,E2 -21888.511} C_VEL
LIN {X 0,Y 307.023,Z 248.514,A -85,B 0,C 180,E1 -21890.198,E2 -21890.198} C_VEL
LIN {X 0,Y 298.783,Z 242.554,A -85,B 0,C 180,E1 -21891.704,E2 -21891.704} C_VEL
LIN {X 0,Y 287.536,Z 233.894,A -85,B 0,C 180,E1 -21893.571,E2 -21893.571} C_VEL
LIN {X 0,Y 273.475,Z 222.368,A -85,B 0,C 180,E1 -21895.915,E2 -21895.915} C_VEL
LIN {X 0,Y 261.209,Z 210.888,A -85,B 0,C 180,E1 -21898.015,E2 -21898.015} C_VEL
LIN {X 0,Y 249.539,Z 198.512,A -85,B 0,C 180,E1 -21900,E2 -21900} C_VEL
LIN {X 0,Y 237.623,Z 183.985,A -85,B 0,C 180,E1 -21902.194,E2 -21902.194} C_VEL
LIN {X 0,Y 228.864,Z 170.632,A -85,B 0,C 180,E1 -21904.091,E2 -21904.091} C_VEL
LIN {X 0,Y 221.937,Z 157.881,A -85,B 0,C 180,E1 -21905.818,E2 -21905.818} C_VEL
LIN {X 0,Y 214.455,Z 142.232,A -85,B 0,C 180,E1 -21907.934,E2 -21907.934} C_VEL
LIN {X 0,Y 207.289,Z 129.253,A -85,B 0,C 180,E1 -21910.08,E2 -21910.08} C_VEL
LIN {X 0,Y 200.3,Z 118.274,A -85,B 0,C 180,E1 -21912.317,E2 -21912.317} C_VEL
LIN {X 0,Y 197.805,Z 114.648,A -85,B 0,C 180,E1 -21913.159,E2 -21913.159} C_VEL
LIN {X 0,Y 195.608,Z 111.162,A -85,B 0,C 180,E1 -21913.945,E2 -21913.945} C_VEL
LIN {X 0,Y 193.393,Z 108.559,A -85,B 0,C 180,E1 -21914.718,E2 -21914.718} C_VEL
LIN {X 0,Y 192.677,Z 106.692,A -85,B 0,C 180,E1 -21915.134,E2 -21915.134} C_VEL
LIN {X 0,Y 192.549,Z 106.036,A -85,B 0,C 180,E1 -21915.722,E2 -21915.722} C_VEL
LIN {X 0,Y 192.541,Z 105.98,A -85,B 0,C 180,E1 -21920.043,E2 -21920.043} C_VEL
LIN {X 0,Y 192.596,Z 105.971,A -85,B 0,C 180,E1 -21924.279,E2 -21924.279} C_VEL
LIN {X 0,Y 192.598,Z 105.995,A -85,B 0,C 180,E1 -21929.28,E2 -21929.28} C_VEL
LIN {X 0,Y 192.659,Z 105.953,A -85,B 0,C 180,E1 -21931.692,E2 -21931.692} C_VEL
LIN {X 0,Y 192.705,Z 105.981,A -85,B 0,C 180,E1 -21936.35,E2 -21936.35} C_VEL
LIN {X 0,Y 192.731,Z 105.933,A -85,B 0,C 180,E1 -21941.459,E2 -21941.459} C_VEL
LIN {X 0,Y 192.772,Z 105.973,A -85,B 0,C 180,E1 -21945.216,E2 -21945.216} C_VEL
LIN {X 0,Y 192.981,Z 105.897,A -85,B 0,C 180,E1 -21949.51,E2 -21949.51} C_VEL
LIN {X 0,Y 193.062,Z 105.893,A -85,B 0,C 180,E1 -21951.628,E2 -21951.628} C_VEL
LIN {X 0,Y 193.264,Z 105.873,A -85,B 0,C 180,E1 -21957.917,E2 -21957.917} C_VEL
LIN {X 0,Y 193.441,Z 105.836,A -85,B 0,C 180,E1 -21960.001,E2 -21960.001} C_VEL
LIN {X 0,Y 192.98,Z 105.944,A -85,B 0,C 180,E1 -21964.178,E2 -21964.178} C_VEL
LIN {X 0,Y 193.064,Z 105.89,A -85,B 0,C 180,E1 -21968.374,E2 -21968.374} C_VEL
LIN {X 0,Y 192.854,Z 105.941,A -85,B 0,C 180,E1 -21972.631,E2 -21972.631} C_VEL
LIN {X 0,Y 192.76,Z 105.937,A -85,B 0,C 180,E1 -21976.96,E2 -21976.96} C_VEL
LIN {X 0,Y 192.638,Z 105.965,A -85,B 0,C 180,E1 -21981.398,E2 -21981.398} C_VEL
LIN {X 0,Y 192.666,Z 105.974,A -85,B 0,C 180,E1 -21984.226,E2 -21984.226} C_VEL
LIN {X 0,Y 192.646,Z 105.962,A -85,B 0,C 180,E1 -21988.89,E2 -21988.89} C_VEL
LIN {X 0,Y 192.598,Z 105.967,A -85,B 0,C 180,E1 -21993.187,E2 -21993.187} C_VEL
LIN {X 0,Y 192.553,Z 105.99,A -85,B 0,C 180,E1 -21998.353,E2 -21998.353} C_VEL
LIN {X 0,Y 192.569,Z 106.13,A -85,B 0,C 180,E1 -22001.91,E2 -22001.91} C_VEL
LIN {X 0,Y 193.544,Z 109.898,A -85,B 0,C 180,E1 -22004.897,E2 -22004.897} C_VEL
LIN {X 0,Y 195.798,Z 114.147,A -85,B 0,C 180,E1 -22005.881,E2 -22005.881} C_VEL
LIN {X 0,Y 200.137,Z 121.606,A -85,B 0,C 180,E1 -22007.422,E2 -22007.422} C_VEL
LIN {X 0,Y 204.988,Z 130.348,A -85,B 0,C 180,E1 -22009.045,E2 -22009.045} C_VEL
LIN {X 0,Y 211.656,Z 144.678,A -85,B 0,C 180,E1 -22011.196,E2 -22011.196} C_VEL
LIN {X 0,Y 215.966,Z 155.674,A -85,B 0,C 180,E1 -22012.555,E2 -22012.555} C_VEL
LIN {X 0,Y 218.389,Z 171.554,A -85,B 0,C 180,E1 -22013.673,E2 -22013.673} C_VEL
LIN {X 0,Y 216.274,Z 216.236,A -85,B 0,C 180,E1 -22015.114,E2 -22015.114} C_VEL
LIN {X 0,Y 215.19,Z 227.22,A -85,B 0,C 180,E1 -22015.678,E2 -22015.678} C_VEL
LIN {X 0,Y 213.627,Z 237.546,A -85,B 0,C 180,E1 -22016.42,E2 -22016.42} C_VEL
LIN {X 0,Y 211.432,Z 249.357,A -85,B 0,C 180,E1 -22017.589,E2 -22017.589} C_VEL
LIN {X 0,Y 208.775,Z 260.751,A -85,B 0,C 180,E1 -22019.112,E2 -22019.112} C_VEL
LIN {X 0,Y 205.884,Z 271.041,A -85,B 0,C 180,E1 -22020.894,E2 -22020.894} C_VEL
LIN {X 0,Y 203.307,Z 279.566,A -85,B 0,C 180,E1 -22022.74,E2 -22022.74} C_VEL
LIN {X 0,Y 200.946,Z 286.782,A -85,B 0,C 180,E1 -22024.632,E2 -22024.632} C_VEL
LIN {X 0,Y 199.282,Z 291.779,A -85,B 0,C 180,E1 -22026.146,E2 -22026.146} C_VEL
LIN {X 0,Y 197.416,Z 295.486,A -85,B 0,C 180,E1 -22027.39,E2 -22027.39} C_VEL
LIN {X 0,Y 192.734,Z 300.999,A -85,B 0,C 180,E1 -22029.376,E2 -22029.376} C_VEL
LIN {X 0,Y 188.143,Z 305.941,A -85,B 0,C 180,E1 -22031.56,E2 -22031.56} C_VEL
LIN {X 0,Y 186.459,Z 308.598,A -85,B 0,C 180,E1 -22033.088,E2 -22033.088} C_VEL
LIN {X 0,Y 185.094,Z 312.408,A -85,B 0,C 180,E1 -22035.712,E2 -22035.712} C_VEL
LIN {X 0,Y 183.976,Z 316.021,A -85,B 0,C 180,E1 -22038.989,E2 -22038.989} C_VEL
LIN {X 0,Y 183.499,Z 317.825,A -85,B 0,C 180,E1 -22041.188,E2 -22041.188} C_VEL
LIN {X 0,Y 183.08,Z 320.281,A -85,B 0,C 180,E1 -22045.597,E2 -22045.597} C_VEL
LIN {X 0,Y 183.05,Z 320.875,A -85,B 0,C 180,E1 -22047.8,E2 -22047.8} C_VEL
LIN {X 0,Y 183.154,Z 321.033,A -85,B 0,C 180,E1 -22050,E2 -22050} C_VEL
LIN {X 0,Y 183.035,Z 320.578,A -85,B 0,C 180,E1 -22053.301,E2 -22053.301} C_VEL
LIN {X 0,Y 183.211,Z 319.218,A -85,B 0,C 180,E1 -22056.608,E2 -22056.608} C_VEL
LIN {X 0,Y 183.499,Z 317.825,A -85,B 0,C 180,E1 -22058.812,E2 -22058.812} C_VEL
LIN {X 0,Y 184.308,Z 314.869,A -85,B 0,C 180,E1 -22062.106,E2 -22062.106} C_VEL
LIN {X 0,Y 185.554,Z 310.875,A -85,B 0,C 180,E1 -22065.375,E2 -22065.375} C_VEL
LIN {X 0,Y 187.573,Z 305.747,A -85,B 0,C 180,E1 -22068.571,E2 -22068.571} C_VEL
LIN {X 0,Y 189.575,Z 300.486,A -85,B 0,C 180,E1 -22071.19,E2 -22071.19} C_VEL
LIN {X 0,Y 191.765,Z 294.547,A -85,B 0,C 180,E1 -22073.617,E2 -22073.617} C_VEL
LIN {X 0,Y 193.966,Z 288.217,A -85,B 0,C 180,E1 -22075.772,E2 -22075.772} C_VEL
LIN {X 0,Y 196.387,Z 281.294,A -85,B 0,C 180,E1 -22077.725,E2 -22077.725} C_VEL
LIN {X 0,Y 199.039,Z 273.119,A -85,B 0,C 180,E1 -22079.626,E2 -22079.626} C_VEL
LIN {X 0,Y 201.57,Z 264.612,A -85,B 0,C 180,E1 -22081.241,E2 -22081.241} C_VEL
LIN {X 0,Y 203.84,Z 255.9,A -85,B 0,C 180,E1 -22082.596,E2 -22082.596} C_VEL
LIN {X 0,Y 206.055,Z 246.146,A -85,B 0,C 180,E1 -22083.805,E2 -22083.805} C_VEL
LIN {X 0,Y 207.971,Z 236.068,A -85,B 0,C 180,E1 -22084.768,E2 -22084.768} C_VEL
LIN {X 0,Y 209.45,Z 225.98,A -85,B 0,C 180,E1 -22085.49,E2 -22085.49} C_VEL
LIN {X 0,Y 210.513,Z 215.821,A -85,B 0,C 180,E1 -22085.994,E2 -22085.994} C_VEL
LIN {X 0,Y 212.624,Z 172.006,A -85,B 0,C 180,E1 -22087.451,E2 -22087.451} C_VEL
LIN {X 0,Y 210.197,Z 157.042,A -85,B 0,C 180,E1 -22088.592,E2 -22088.592} C_VEL
LIN {X 0,Y 204.041,Z 142.404,A -85,B 0,C 180,E1 -22090.636,E2 -22090.636} C_VEL
LIN {X 0,Y 198.812,Z 131.701,A -85,B 0,C 180,E1 -22092.443,E2 -22092.443} C_VEL
LIN {X 0,Y 194.062,Z 123.106,A -85,B 0,C 180,E1 -22094.162,E2 -22094.162} C_VEL
LIN {X 0,Y 189.09,Z 114.516,A -85,B 0,C 180,E1 -22096.091,E2 -22096.091} C_VEL
LIN {X 0,Y 186.459,Z 110.362,A -85,B 0,C 180,E1 -22097.203,E2 -22097.203} C_VEL
LIN {X 0,Y 186.018,Z 109.058,A -85,B 0,C 180,E1 -22097.772,E2 -22097.772} C_VEL
LIN {X 0,Y 185.472,Z 106.881,A -85,B 0,C 180,E1 -22099.895,E2 -22099.895} C_VEL
LIN {X 0,Y 185.51,Z 106.878,A -85,B 0,C 180,E1 -22102.71,E2 -22102.71} C_VEL
LIN {X 0,Y 185.544,Z 106.859,A -85,B 0,C 180,E1 -22107.974,E2 -22107.974} C_VEL
LIN {X 0,Y 185.582,Z 106.849,A -85,B 0,C 180,E1 -22110.576,E2 -22110.576} C_VEL
LIN {X 0,Y 185.589,Z 106.847,A -85,B 0,C 180,E1 -22115.382,E2 -22115.382} C_VEL
LIN {X 0,Y 185.609,Z 106.82,A -85,B 0,C 180,E1 -22120.074,E2 -22120.074} C_VEL
LIN {X 0,Y 185.726,Z 106.84,A -85,B 0,C 180,E1 -22124.639,E2 -22124.639} C_VEL
LIN {X 0,Y 185.925,Z 106.775,A -85,B 0,C 180,E1 -22129.358,E2 -22129.358} C_VEL
LIN {X 0,Y 185.963,Z 106.803,A -85,B 0,C 180,E1 -22133.489,E2 -22133.489} C_VEL
LIN {X 0,Y 186.209,Z 106.754,A -85,B 0,C 180,E1 -22137.836,E2 -22137.836} C_VEL
LIN {X 0,Y 186.405,Z 106.712,A -85,B 0,C 180,E1 -22139.999,E2 -22139.999} C_VEL
LIN {X 0,Y 185.926,Z 106.822,A -85,B 0,C 180,E1 -22144.335,E2 -22144.335} C_VEL
LIN {X 0,Y 186.009,Z 106.767,A -85,B 0,C 180,E1 -22148.691,E2 -22148.691} C_VEL
LIN {X 0,Y 185.765,Z 106.831,A -85,B 0,C 180,E1 -22153.119,E2 -22153.119} C_VEL
LIN {X 0,Y 185.69,Z 106.815,A -85,B 0,C 180,E1 -22157.624,E2 -22157.624} C_VEL
LIN {X 0,Y 185.596,Z 106.857,A -85,B 0,C 180,E1 -22162.25,E2 -22162.25} C_VEL
LIN {X 0,Y 185.559,Z 106.833,A -85,B 0,C 180,E1 -22167.031,E2 -22167.031} C_VEL
LIN {X 0,Y 185.576,Z 106.848,A -85,B 0,C 180,E1 -22169.492,E2 -22169.492} C_VEL
LIN {X 0,Y 185.516,Z 106.847,A -85,B 0,C 180,E1 -22174.627,E2 -22174.627} C_VEL
LIN {X 0,Y 185.542,Z 106.872,A -85,B 0,C 180,E1 -22177.303,E2 -22177.303} C_VEL
LIN {X 0,Y 185.463,Z 106.968,A -85,B 0,C 180,E1 -22182.23,E2 -22182.23} C_VEL
LIN {X 0,Y 185.689,Z 107.962,A -85,B 0,C 180,E1 -22182.785,E2 -22182.785} C_VEL
LIN {X 0,Y 187.305,Z 110.789,A -85,B 0,C 180,E1 -22183.516,E2 -22183.516} C_VEL
LIN {X 0,Y 188.839,Z 112.38,A -85,B 0,C 180,E1 -22184.093,E2 -22184.093} C_VEL
LIN {X 0,Y 191.072,Z 115.81,A -85,B 0,C 180,E1 -22184.964,E2 -22184.964} C_VEL
LIN {X 0,Y 197.345,Z 124.926,A -85,B 0,C 180,E1 -22187.217,E2 -22187.217} C_VEL
LIN {X 0,Y 205.077,Z 137.742,A -85,B 0,C 180,E1 -22189.778,E2 -22189.778} C_VEL
LIN {X 0,Y 212.777,Z 152.752,A -85,B 0,C 180,E1 -22192.154,E2 -22192.154} C_VEL
LIN {X 0,Y 221.233,Z 170.317,A -85,B 0,C 180,E1 -22194.538,E2 -22194.538} C_VEL
LIN {X 0,Y 229.69,Z 184.067,A -85,B 0,C 180,E1 -22196.545,E2 -22196.545} C_VEL
LIN {X 0,Y 238.157,Z 195.494,A -85,B 0,C 180,E1 -22198.288,E2 -22198.288} C_VEL
LIN {X 0,Y 248.488,Z 207.563,A -85,B 0,C 180,E1 -22200.218,E2 -22200.218} C_VEL
LIN {X 0,Y 260.324,Z 219.934,A -85,B 0,C 180,E1 -22202.458,E2 -22202.458} C_VEL
LIN {X 0,Y 272.186,Z 230.612,A -85,B 0,C 180,E1 -22204.649,E2 -22204.649} C_VEL
LIN {X 0,Y 284.679,Z 240.558,A -85,B 0,C 180,E1 -22206.866,E2 -22206.866} C_VEL
LIN {X 0,Y 297.224,Z 250.018,A -85,B 0,C 180,E1 -22209.066,E2 -22209.066} C_VEL
LIN {X 0,Y 304.452,Z 255.319,A -85,B 0,C 180,E1 -22210.45,E2 -22210.45} C_VEL
LIN {X 0,Y 310.727,Z 259.81,A -85,B 0,C 180,E1 -22211.794,E2 -22211.794} C_VEL
LIN {X 0,Y 316.846,Z 264.046,A -85,B 0,C 180,E1 -22213.241,E2 -22213.241} C_VEL
LIN {X 0,Y 322.724,Z 268.269,A -85,B 0,C 180,E1 -22214.851,E2 -22214.851} C_VEL
LIN {X 0,Y 327.87,Z 271.504,A -85,B 0,C 180,E1 -22216.362,E2 -22216.362} C_VEL
LIN {X 0,Y 332.224,Z 274.178,A -85,B 0,C 180,E1 -22217.787,E2 -22217.787} C_VEL
LIN {X 0,Y 336.066,Z 276.973,A -85,B 0,C 180,E1 -22219.382,E2 -22219.382} C_VEL
LIN {X 0,Y 338.409,Z 278.534,A -85,B 0,C 180,E1 -22220.436,E2 -22220.436} C_VEL
LIN {X 0,Y 340.969,Z 280.065,A -85,B 0,C 180,E1 -22221.704,E2 -22221.704} C_VEL
LIN {X 0,Y 343.175,Z 281.305,A -85,B 0,C 180,E1 -22222.942,E2 -22222.942} C_VEL
LIN {X 0,Y 345.849,Z 282.504,A -85,B 0,C 180,E1 -22224.694,E2 -22224.694} C_VEL
LIN {X 0,Y 347.928,Z 283.298,A -85,B 0,C 180,E1 -22226.526,E2 -22226.526} C_VEL
LIN {X 0,Y 348.767,Z 283.64,A -85,B 0,C 180,E1 -22227.69,E2 -22227.69} C_VEL
LIN {X 0,Y 349.163,Z 283.93,A -85,B 0,C 180,E1 -22228.847,E2 -22228.847} C_VEL
LIN {X 0,Y 349.387,Z 283.937,A -85,B 0,C 180,E1 -22230,E2 -22230} C_VEL
LIN {X 0,Y 349.212,Z 283.872,A -85,B 0,C 180,E1 -22231.153,E2 -22231.153} C_VEL
LIN {X 0,Y 348.771,Z 283.61,A -85,B 0,C 180,E1 -22232.31,E2 -22232.31} C_VEL
LIN {X 0,Y 347.949,Z 283.246,A -85,B 0,C 180,E1 -22233.474,E2 -22233.474} C_VEL
LIN {X 0,Y 345.849,Z 282.544,A -85,B 0,C 180,E1 -22235.306,E2 -22235.306} C_VEL
LIN {X 0,Y 343.163,Z 281.283,A -85,B 0,C 180,E1 -22237.058,E2 -22237.058} C_VEL
LIN {X 0,Y 340.916,Z 280.062,A -85,B 0,C 180,E1 -22238.306,E2 -22238.306} C_VEL
LIN {X 0,Y 338.404,Z 278.511,A -85,B 0,C 180,E1 -22239.564,E2 -22239.564} C_VEL
LIN {X 0,Y 335.474,Z 276.554,A -85,B 0,C 180,E1 -22240.868,E2 -22240.868} C_VEL
LIN {X 0,Y 331.234,Z 273.486,A -85,B 0,C 180,E1 -22242.579,E2 -22242.579} C_VEL
LIN {X 0,Y 325.213,Z 269.847,A -85,B 0,C 180,E1 -22244.442,E2 -22244.442} C_VEL
LIN {X 0,Y 318.528,Z 265.287,A -85,B 0,C 180,E1 -22246.31,E2 -22246.31} C_VEL
LIN {X 0,Y 313.268,Z 261.526,A -85,B 0,C 180,E1 -22247.638,E2 -22247.638} C_VEL
LIN {X 0,Y 305.394,Z 256.083,A -85,B 0,C 180,E1 -22249.35,E2 -22249.35} C_VEL
LIN {X 0,Y 298.804,Z 251.104,A -85,B 0,C 180,E1 -22250.659,E2 -22250.659} C_VEL
LIN {X 0,Y 286.084,Z 241.579,A -85,B 0,C 180,E1 -22252.895,E2 -22252.895} C_VEL
LIN {X 0,Y 273.572,Z 231.752,A -85,B 0,C 180,E1 -22255.103,E2 -22255.103} C_VEL
LIN {X 0,Y 259.986,Z 219.575,A -85,B 0,C 180,E1 -22257.609,E2 -22257.609} C_VEL
LIN {X 0,Y 248.492,Z 207.526,A -85,B 0,C 180,E1 -22259.784,E2 -22259.784} C_VEL
LIN {X 0,Y 237.053,Z 194.182,A -85,B 0,C 180,E1 -22261.924,E2 -22261.924} C_VEL
LIN {X 0,Y 227.608,Z 180.989,A -85,B 0,C 180,E1 -22263.92,E2 -22263.92} C_VEL
LIN {X 0,Y 219.551,Z 167.061,A -85,B 0,C 180,E1 -22265.907,E2 -22265.907} C_VEL
LIN {X 0,Y 209.209,Z 145.548,A -85,B 0,C 180,E1 -22268.926,E2 -22268.926} C_VEL
LIN {X 0,Y 202.597,Z 133.429,A -85,B 0,C 180,E1 -22271.021,E2 -22271.021} C_VEL
LIN {X 0,Y 195.705,Z 122.549,A -85,B 0,C 180,E1 -22273.349,E2 -22273.349} C_VEL
LIN {X 0,Y 191.073,Z 115.804,A -85,B 0,C 180,E1 -22275.036,E2 -22275.036} C_VEL
LIN {X 0,Y 188.932,Z 112.565,A -85,B 0,C 180,E1 -22275.867,E2 -22275.867} C_VEL
LIN {X 0,Y 188.133,Z 111.551,A -85,B 0,C 180,E1 -22276.176,E2 -22276.176} C_VEL
LIN {X 0,Y 186.355,Z 109.467,A -85,B 0,C 180,E1 -22276.867,E2 -22276.867} C_VEL
LIN {X 0,Y 185.595,Z 107.553,A -85,B 0,C 180,E1 -22277.343,E2 -22277.343} C_VEL
LIN {X 0,Y 185.474,Z 106.915,A -85,B 0,C 180,E1 -22277.927,E2 -22277.927} C_VEL
LIN {X 0,Y 185.542,Z 106.872,A -85,B 0,C 180,E1 -22282.697,E2 -22282.697} C_VEL
LIN {X 0,Y 185.539,Z 106.864,A -85,B 0,C 180,E1 -22287.975,E2 -22287.975} C_VEL
LIN {X 0,Y 185.579,Z 106.847,A -85,B 0,C 180,E1 -22290.578,E2 -22290.578} C_VEL
LIN {X 0,Y 185.586,Z 106.854,A -85,B 0,C 180,E1 -22295.384,E2 -22295.384} C_VEL
LIN {X 0,Y 185.606,Z 106.822,A -85,B 0,C 180,E1 -22300.077,E2 -22300.077} C_VEL
LIN {X 0,Y 185.724,Z 106.846,A -85,B 0,C 180,E1 -22304.641,E2 -22304.641} C_VEL
LIN {X 0,Y 185.924,Z 106.776,A -85,B 0,C 180,E1 -22309.36,E2 -22309.36} C_VEL
LIN {X 0,Y 185.962,Z 106.806,A -85,B 0,C 180,E1 -22313.491,E2 -22313.491} C_VEL
LIN {X 0,Y 186.208,Z 106.751,A -85,B 0,C 180,E1 -22317.838,E2 -22317.838} C_VEL
LIN {X 0,Y 186.405,Z 106.712,A -85,B 0,C 180,E1 -22320.001,E2 -22320.001} C_VEL
LIN {X 0,Y 185.927,Z 106.824,A -85,B 0,C 180,E1 -22324.337,E2 -22324.337} C_VEL
LIN {X 0,Y 186.01,Z 106.765,A -85,B 0,C 180,E1 -22328.694,E2 -22328.694} C_VEL
LIN {X 0,Y 185.766,Z 106.831,A -85,B 0,C 180,E1 -22333.121,E2 -22333.121} C_VEL
LIN {X 0,Y 185.692,Z 106.81,A -85,B 0,C 180,E1 -22337.626,E2 -22337.626} C_VEL
LIN {X 0,Y 185.599,Z 106.857,A -85,B 0,C 180,E1 -22342.252,E2 -22342.252} C_VEL
LIN {X 0,Y 185.562,Z 106.831,A -85,B 0,C 180,E1 -22347.033,E2 -22347.033} C_VEL
LIN {X 0,Y 185.579,Z 106.851,A -85,B 0,C 180,E1 -22349.494,E2 -22349.494} C_VEL
LIN {X 0,Y 185.501,Z 106.847,A -85,B 0,C 180,E1 -22354.633,E2 -22354.633} C_VEL
LIN {X 0,Y 185.509,Z 106.878,A -85,B 0,C 180,E1 -22357.314,E2 -22357.314} C_VEL
LIN {X 0,Y 185.494,Z 106.948,A -85,B 0,C 180,E1 -22360.318,E2 -22360.318} C_VEL
LIN {X 0,Y 186.134,Z 109.49,A -85,B 0,C 180,E1 -22362.505,E2 -22362.505} C_VEL
LIN {X 0,Y 187.806,Z 112.861,A -85,B 0,C 180,E1 -22363.414,E2 -22363.414} C_VEL
LIN {X 0,Y 189.925,Z 115.902,A -85,B 0,C 180,E1 -22364.242,E2 -22364.242} C_VEL
LIN {X 0,Y 196.433,Z 127.322,A -85,B 0,C 180,E1 -22366.709,E2 -22366.709} C_VEL
LIN {X 0,Y 201.285,Z 136.415,A -85,B 0,C 180,E1 -22368.413,E2 -22368.413} C_VEL
LIN {X 0,Y 208.17,Z 152.023,A -85,B 0,C 180,E1 -22370.746,E2 -22370.746} C_VEL
LIN {X 0,Y 210.537,Z 158.283,A -85,B 0,C 180,E1 -22371.534,E2 -22371.534} C_VEL
LIN {X 0,Y 212.667,Z 172.706,A -85,B 0,C 180,E1 -22372.587,E2 -22372.587} C_VEL
LIN {X 0,Y 210.444,Z 216.809,A -85,B 0,C 180,E1 -22374.044,E2 -22374.044} C_VEL
LIN {X 0,Y 209.188,Z 228.564,A -85,B 0,C 180,E1 -22374.677,E2 -22374.677} C_VEL
LIN {X 0,Y 206.909,Z 242.12,A -85,B 0,C 180,E1 -22375.766,E2 -22375.766} C_VEL
LIN {X 0,Y 204.617,Z 252.637,A -85,B 0,C 180,E1 -22376.958,E2 -22376.958} C_VEL
LIN {X 0,Y 202.304,Z 261.91,A -85,B 0,C 180,E1 -22378.302,E2 -22378.302} C_VEL
LIN {X 0,Y 199.691,Z 270.849,A -85,B 0,C 180,E1 -22379.899,E2 -22379.899} C_VEL
LIN {X 0,Y 197.013,Z 279.375,A -85,B 0,C 180,E1 -22381.793,E2 -22381.793} C_VEL
LIN {X 0,Y 194.536,Z 286.591,A -85,B 0,C 180,E1 -22383.733,E2 -22383.733} C_VEL
LIN {X 0,Y 192.332,Z 292.791,A -85,B 0,C 180,E1 -22385.727,E2 -22385.727} C_VEL
LIN {X 0,Y 190.039,Z 299.331,A -85,B 0,C 180,E1 -22388.296,E2 -22388.296} C_VEL
LIN {X 0,Y 188.316,Z 303.831,A -85,B 0,C 180,E1 -22390.374,E2 -22390.374} C_VEL
LIN {X 0,Y 186.459,Z 308.598,A -85,B 0,C 180,E1 -22393.088,E2 -22393.088} C_VEL
LIN {X 0,Y 184.895,Z 311.056,A -85,B 0,C 180,E1 -22394.685,E2 -22394.685} C_VEL
LIN {X 0,Y 180.895,Z 314.412,A -85,B 0,C 180,E1 -22397.325,E2 -22397.325} C_VEL
LIN {X 0,Y 177.83,Z 316.611,A -85,B 0,C 180,E1 -22399.562,E2 -22399.562} C_VEL
LIN {X 0,Y 176.328,Z 318.266,A -85,B 0,C 180,E1 -22401.684,E2 -22401.684} C_VEL
LIN {X 0,Y 176.261,Z 318.342,A -85,B 0,C 180,E1 -22401.997,E2 -22401.997} C_VEL
LIN {X 0,Y 176.01,Z 320.091,A -85,B 0,C 180,E1 -22405.42,E2 -22405.42} C_VEL
LIN {X 0,Y 175.972,Z 320.685,A -85,B 0,C 180,E1 -22407.711,E2 -22407.711} C_VEL
LIN {X 0,Y 176.062,Z 320.843,A -85,B 0,C 180,E1 -22410,E2 -22410} C_VEL
LIN {X 0,Y 175.95,Z 320.491,A -85,B 0,C 180,E1 -22413.037,E2 -22413.037} C_VEL
LIN {X 0,Y 176.139,Z 319.027,A -85,B 0,C 180,E1 -22416.875,E2 -22416.875} C_VEL
LIN {X 0,Y 176.459,Z 317.634,A -85,B 0,C 180,E1 -22419.167,E2 -22419.167} C_VEL
LIN {X 0,Y 177.335,Z 314.678,A -85,B 0,C 180,E1 -22422.59,E2 -22422.59} C_VEL
LIN {X 0,Y 178.69,Z 310.684,A -85,B 0,C 180,E1 -22425.981,E2 -22425.981} C_VEL
LIN {X 0,Y 180.834,Z 305.556,A -85,B 0,C 180,E1 -22429.29,E2 -22429.29} C_VEL
LIN {X 0,Y 182.969,Z 300.295,A -85,B 0,C 180,E1 -22431.994,E2 -22431.994} C_VEL
LIN {X 0,Y 185.4,Z 293.978,A -85,B 0,C 180,E1 -22434.644,E2 -22434.644} C_VEL
LIN {X 0,Y 187.574,Z 288.026,A -85,B 0,C 180,E1 -22436.719,E2 -22436.719} C_VEL
LIN {X 0,Y 190.105,Z 281.103,A -85,B 0,C 180,E1 -22438.724,E2 -22438.724} C_VEL
LIN {X 0,Y 192.875,Z 272.928,A -85,B 0,C 180,E1 -22440.673,E2 -22440.673} C_VEL
LIN {X 0,Y 195.53,Z 264.422,A -85,B 0,C 180,E1 -22442.321,E2 -22442.321} C_VEL
LIN {X 0,Y 197.894,Z 255.71,A -85,B 0,C 180,E1 -22443.704,E2 -22443.704} C_VEL
LIN {X 0,Y 200.204,Z 245.956,A -85,B 0,C 180,E1 -22444.934,E2 -22444.934} C_VEL
LIN {X 0,Y 202.186,Z 235.878,A -85,B 0,C 180,E1 -22445.914,E2 -22445.914} C_VEL
LIN {X 0,Y 203.739,Z 225.567,A -85,B 0,C 180,E1 -22446.663,E2 -22446.663} C_VEL
LIN {X 0,Y 204.785,Z 215.894,A -85,B 0,C 180,E1 -22447.151,E2 -22447.151} C_VEL
LIN {X 0,Y 207.002,Z 173.341,A -85,B 0,C 180,E1 -22448.587,E2 -22448.587} C_VEL
LIN {X 0,Y 204.921,Z 159.937,A -85,B 0,C 180,E1 -22449.643,E2 -22449.643} C_VEL
LIN {X 0,Y 198.839,Z 145.359,A -85,B 0,C 180,E1 -22451.787,E2 -22451.787} C_VEL
LIN {X 0,Y 193,Z 133.349,A -85,B 0,C 180,E1 -22453.947,E2 -22453.947} C_VEL
LIN {X 0,Y 186.928,Z 122.711,A -85,B 0,C 180,E1 -22456.332,E2 -22456.332} C_VEL
LIN {X 0,Y 184.745,Z 119.001,A -85,B 0,C 180,E1 -22457.248,E2 -22457.248} C_VEL
LIN {X 0,Y 181.648,Z 114.086,A -85,B 0,C 180,E1 -22458.595,E2 -22458.595} C_VEL
LIN {X 0,Y 179.19,Z 110.206,A -85,B 0,C 180,E1 -22459.764,E2 -22459.764} C_VEL
LIN {X 0,Y 178.688,Z 109.005,A -85,B 0,C 180,E1 -22460.271,E2 -22460.271} C_VEL
LIN {X 0,Y 178.411,Z 107.791,A -85,B 0,C 180,E1 -22461.55,E2 -22461.55} C_VEL
LIN {X 0,Y 178.487,Z 107.722,A -85,B 0,C 180,E1 -22466.546,E2 -22466.546} C_VEL
LIN {X 0,Y 178.523,Z 107.737,A -85,B 0,C 180,E1 -22470.006,E2 -22470.006} C_VEL
LIN {X 0,Y 178.526,Z 107.718,A -85,B 0,C 180,E1 -22474.882,E2 -22474.882} C_VEL
LIN {X 0,Y 178.625,Z 107.685,A -85,B 0,C 180,E1 -22480.783,E2 -22480.783} C_VEL
LIN {X 0,Y 178.667,Z 107.705,A -85,B 0,C 180,E1 -22484.016,E2 -22484.016} C_VEL
LIN {X 0,Y 178.862,Z 107.654,A -85,B 0,C 180,E1 -22489.209,E2 -22489.209} C_VEL
LIN {X 0,Y 178.927,Z 107.672,A -85,B 0,C 180,E1 -22493.232,E2 -22493.232} C_VEL
LIN {X 0,Y 179.155,Z 107.632,A -85,B 0,C 180,E1 -22497.751,E2 -22497.751} C_VEL
LIN {X 0,Y 179.369,Z 107.587,A -85,B 0,C 180,E1 -22499.999,E2 -22499.999} C_VEL
LIN {X 0,Y 178.874,Z 107.702,A -85,B 0,C 180,E1 -22504.506,E2 -22504.506} C_VEL
LIN {X 0,Y 178.938,Z 107.645,A -85,B 0,C 180,E1 -22509.038,E2 -22509.038} C_VEL
LIN {X 0,Y 178.687,Z 107.721,A -85,B 0,C 180,E1 -22513.649,E2 -22513.649} C_VEL
LIN {X 0,Y 178.649,Z 107.686,A -85,B 0,C 180,E1 -22518.342,E2 -22518.342} C_VEL
LIN {X 0,Y 178.511,Z 107.75,A -85,B 0,C 180,E1 -22523.184,E2 -22523.184} C_VEL
LIN {X 0,Y 178.483,Z 107.717,A -85,B 0,C 180,E1 -22528.196,E2 -22528.196} C_VEL
LIN {X 0,Y 178.496,Z 107.752,A -85,B 0,C 180,E1 -22530.786,E2 -22530.786} C_VEL
LIN {X 0,Y 178.493,Z 107.721,A -85,B 0,C 180,E1 -22534.223,E2 -22534.223} C_VEL
LIN {X 0,Y 178.477,Z 107.9,A -85,B 0,C 180,E1 -22539.782,E2 -22539.782} C_VEL
LIN {X 0,Y 178.718,Z 108.928,A -85,B 0,C 180,E1 -22540.361,E2 -22540.361} C_VEL
LIN {X 0,Y 180.207,Z 111.597,A -85,B 0,C 180,E1 -22541.116,E2 -22541.116} C_VEL
LIN {X 0,Y 181.86,Z 113.189,A -85,B 0,C 180,E1 -22541.806,E2 -22541.806} C_VEL
LIN {X 0,Y 184.05,Z 116.628,A -85,B 0,C 180,E1 -22542.762,E2 -22542.762} C_VEL
LIN {X 0,Y 185.408,Z 118.324,A -85,B 0,C 180,E1 -22543.311,E2 -22543.311} C_VEL
LIN {X 0,Y 193.106,Z 129.657,A -85,B 0,C 180,E1 -22546.274,E2 -22546.274} C_VEL
LIN {X 0,Y 200.712,Z 142.481,A -85,B 0,C 180,E1 -22548.93,E2 -22548.93} C_VEL
LIN {X 0,Y 208.287,Z 157.585,A -85,B 0,C 180,E1 -22551.391,E2 -22551.391} C_VEL
LIN {X 0,Y 216.236,Z 174.356,A -85,B 0,C 180,E1 -22553.746,E2 -22553.746} C_VEL
LIN {X 0,Y 225.067,Z 188.887,A -85,B 0,C 180,E1 -22555.94,E2 -22555.94} C_VEL
LIN {X 0,Y 233.642,Z 200.579,A -85,B 0,C 180,E1 -22557.778,E2 -22557.778} C_VEL
LIN {X 0,Y 243.793,Z 212.656,A -85,B 0,C 180,E1 -22559.861,E2 -22559.861} C_VEL
LIN {X 0,Y 254.498,Z 224.041,A -85,B 0,C 180,E1 -22562.088,E2 -22562.088} C_VEL
LIN {X 0,Y 266.625,Z 235.175,A -85,B 0,C 180,E1 -22564.526,E2 -22564.526} C_VEL
LIN {X 0,Y 279.939,Z 245.748,A -85,B 0,C 180,E1 -22567.06,E2 -22567.06} C_VEL
LIN {X 0,Y 292.757,Z 255.209,A -85,B 0,C 180,E1 -22569.428,E2 -22569.428} C_VEL
LIN {X 0,Y 300.111,Z 260.636,A -85,B 0,C 180,E1 -22570.862,E2 -22570.862} C_VEL
LIN {X 0,Y 307.409,Z 265.749,A -85,B 0,C 180,E1 -22572.425,E2 -22572.425} C_VEL
LIN {X 0,Y 314.19,Z 270.62,A -85,B 0,C 180,E1 -22574.12,E2 -22574.12} C_VEL
LIN {X 0,Y 321.062,Z 275.202,A -85,B 0,C 180,E1 -22576.067,E2 -22576.067} C_VEL
LIN {X 0,Y 325.811,Z 278.039,A -85,B 0,C 180,E1 -22577.543,E2 -22577.543} C_VEL
LIN {X 0,Y 331.104,Z 281.835,A -85,B 0,C 180,E1 -22579.674,E2 -22579.674} C_VEL
LIN {X 0,Y 335.084,Z 284.361,A -85,B 0,C 180,E1 -22581.558,E2 -22581.558} C_VEL
LIN {X 0,Y 337.383,Z 285.68,A -85,B 0,C 180,E1 -22582.82,E2 -22582.82} C_VEL
LIN {X 0,Y 339.401,Z 286.652,A -85,B 0,C 180,E1 -22584.057,E2 -22584.057} C_VEL
LIN {X 0,Y 341.088,Z 287.373,A -85,B 0,C 180,E1 -22585.272,E2 -22585.272} C_VEL
LIN {X 0,Y 342.421,Z 287.868,A -85,B 0,C 180,E1 -22586.47,E2 -22586.47} C_VEL
LIN {X 0,Y 343.32,Z 288.214,A -85,B 0,C 180,E1 -22587.654,E2 -22587.654} C_VEL
LIN {X 0,Y 343.742,Z 288.502,A -85,B 0,C 180,E1 -22588.828,E2 -22588.828} C_VEL
LIN {X 0,Y 343.979,Z 288.514,A -85,B 0,C 180,E1 -22590,E2 -22590} C_VEL
LIN {X 0,Y 343.793,Z 288.447,A -85,B 0,C 180,E1 -22591.171,E2 -22591.171} C_VEL
LIN {X 0,Y 343.323,Z 288.189,A -85,B 0,C 180,E1 -22592.346,E2 -22592.346} C_VEL
LIN {X 0,Y 342.437,Z 287.826,A -85,B 0,C 180,E1 -22593.53,E2 -22593.53} C_VEL
LIN {X 0,Y 341.054,Z 287.363,A -85,B 0,C 180,E1 -22594.728,E2 -22594.728} C_VEL
LIN {X 0,Y 339.224,Z 286.565,A -85,B 0,C 180,E1 -22596.043,E2 -22596.043} C_VEL
LIN {X 0,Y 337.368,Z 285.666,A -85,B 0,C 180,E1 -22597.18,E2 -22597.18} C_VEL
LIN {X 0,Y 334.285,Z 283.895,A -85,B 0,C 180,E1 -22598.843,E2 -22598.843} C_VEL
LIN {X 0,Y 331.125,Z 281.845,A -85,B 0,C 180,E1 -22600.318,E2 -22600.318} C_VEL
LIN {X 0,Y 325.811,Z 278.028,A -85,B 0,C 180,E1 -22602.457,E2 -22602.457} C_VEL
LIN {X 0,Y 319.315,Z 274.111,A -85,B 0,C 180,E1 -22604.44,E2 -22604.44} C_VEL
LIN {X 0,Y 314.19,Z 270.622,A -85,B 0,C 180,E1 -22605.88,E2 -22605.88} C_VEL
LIN {X 0,Y 307.406,Z 265.783,A -85,B 0,C 180,E1 -22607.573,E2 -22607.573} C_VEL
LIN {X 0,Y 300.073,Z 260.672,A -85,B 0,C 180,E1 -22609.141,E2 -22609.141} C_VEL
LIN {X 0,Y 292.751,Z 255.235,A -85,B 0,C 180,E1 -22610.569,E2 -22610.569} C_VEL
LIN {X 0,Y 278.052,Z 244.35,A -85,B 0,C 180,E1 -22613.289,E2 -22613.289} C_VEL
LIN {X 0,Y 265.274,Z 233.996,A -85,B 0,C 180,E1 -22615.742,E2 -22615.742} C_VEL
LIN {X 0,Y 253.507,Z 223.072,A -85,B 0,C 180,E1 -22618.118,E2 -22618.118} C_VEL
LIN {X 0,Y 242.29,Z 210.876,A -85,B 0,C 180,E1 -22620.456,E2 -22620.456} C_VEL
LIN {X 0,Y 232.442,Z 199.108,A -85,B 0,C 180,E1 -22622.463,E2 -22622.463} C_VEL
LIN {X 0,Y 222.769,Z 185.448,A -85,B 0,C 180,E1 -22624.595,E2 -22624.595} C_VEL
LIN {X 0,Y 215.027,Z 171.963,A -85,B 0,C 180,E1 -22626.59,E2 -22626.59} C_VEL
LIN {X 0,Y 204.612,Z 150.008,A -85,B 0,C 180,E1 -22629.78,E2 -22629.78} C_VEL
LIN {X 0,Y 198.012,Z 137.726,A -85,B 0,C 180,E1 -22631.987,E2 -22631.987} C_VEL
LIN {X 0,Y 191.511,Z 127.321,A -85,B 0,C 180,E1 -22634.308,E2 -22634.308} C_VEL
LIN {X 0,Y 186.885,Z 120.567,A -85,B 0,C 180,E1 -22636.085,E2 -22636.085} C_VEL
LIN {X 0,Y 184.458,Z 117.06,A -85,B 0,C 180,E1 -22637.076,E2 -22637.076} C_VEL
LIN {X 0,Y 182.104,Z 113.714,A -85,B 0,C 180,E1 -22638.077,E2 -22638.077} C_VEL
LIN {X 0,Y 181.329,Z 112.628,A -85,B 0,C 180,E1 -22638.416,E2 -22638.416} C_VEL
LIN {X 0,Y 179.303,Z 110.343,A -85,B 0,C 180,E1 -22639.294,E2 -22639.294} C_VEL
LIN {X 0,Y 178.556,Z 108.311,A -85,B 0,C 180,E1 -22639.872,E2 -22639.872} C_VEL
LIN {X 0,Y 178.438,Z 107.786,A -85,B 0,C 180,E1 -22640.574,E2 -22640.574} C_VEL
LIN {X 0,Y 178.493,Z 107.721,A -85,B 0,C 180,E1 -22645.777,E2 -22645.777} C_VEL
LIN {X 0,Y 178.52,Z 107.734,A -85,B 0,C 180,E1 -22650.008,E2 -22650.008} C_VEL
LIN {X 0,Y 178.533,Z 107.723,A -85,B 0,C 180,E1 -22654.877,E2 -22654.877} C_VEL
LIN {X 0,Y 178.622,Z 107.688,A -85,B 0,C 180,E1 -22660.785,E2 -22660.785} C_VEL
LIN {X 0,Y 178.665,Z 107.714,A -85,B 0,C 180,E1 -22664.018,E2 -22664.018} C_VEL
LIN {X 0,Y 178.861,Z 107.656,A -85,B 0,C 180,E1 -22669.211,E2 -22669.211} C_VEL
LIN {X 0,Y 178.925,Z 107.676,A -85,B 0,C 180,E1 -22673.234,E2 -22673.234} C_VEL
LIN {X 0,Y 179.154,Z 107.629,A -85,B 0,C 180,E1 -22677.753,E2 -22677.753} C_VEL
LIN {X 0,Y 179.369,Z 107.587,A -85,B 0,C 180,E1 -22680.001,E2 -22680.001} C_VEL
LIN {X 0,Y 178.876,Z 107.704,A -85,B 0,C 180,E1 -22684.508,E2 -22684.508} C_VEL
LIN {X 0,Y 178.939,Z 107.642,A -85,B 0,C 180,E1 -22689.04,E2 -22689.04} C_VEL
LIN {X 0,Y 178.689,Z 107.72,A -85,B 0,C 180,E1 -22693.651,E2 -22693.651} C_VEL
LIN {X 0,Y 178.652,Z 107.682,A -85,B 0,C 180,E1 -22698.345,E2 -22698.345} C_VEL
LIN {X 0,Y 178.514,Z 107.747,A -85,B 0,C 180,E1 -22703.186,E2 -22703.186} C_VEL
LIN {X 0,Y 178.487,Z 107.716,A -85,B 0,C 180,E1 -22708.198,E2 -22708.198} C_VEL
LIN {X 0,Y 178.501,Z 107.751,A -85,B 0,C 180,E1 -22710.788,E2 -22710.788} C_VEL
LIN {X 0,Y 178.486,Z 107.72,A -85,B 0,C 180,E1 -22714.22,E2 -22714.22} C_VEL
LIN {X 0,Y 178.425,Z 107.934,A -85,B 0,C 180,E1 -22718.757,E2 -22718.757} C_VEL
LIN {X 0,Y 178.91,Z 109.579,A -85,B 0,C 180,E1 -22720.036,E2 -22720.036} C_VEL
LIN {X 0,Y 181.256,Z 113.599,A -85,B 0,C 180,E1 -22721.237,E2 -22721.237} C_VEL
LIN {X 0,Y 182.929,Z 116.103,A -85,B 0,C 180,E1 -22721.971,E2 -22721.971} C_VEL
LIN {X 0,Y 186.196,Z 121.35,A -85,B 0,C 180,E1 -22723.358,E2 -22723.358} C_VEL
LIN {X 0,Y 192.129,Z 131.85,A -85,B 0,C 180,E1 -22725.727,E2 -22725.727} C_VEL
LIN {X 0,Y 197.035,Z 141.36,A -85,B 0,C 180,E1 -22727.553,E2 -22727.553} C_VEL
LIN {X 0,Y 203.162,Z 155.553,A -85,B 0,C 180,E1 -22729.75,E2 -22729.75} C_VEL
LIN {X 0,Y 205.198,Z 160.948,A -85,B 0,C 180,E1 -22730.466,E2 -22730.466} C_VEL
LIN {X 0,Y 207.014,Z 173.961,A -85,B 0,C 180,E1 -22731.443,E2 -22731.443} C_VEL
LIN {X 0,Y 204.795,Z 216.03,A -85,B 0,C 180,E1 -22732.852,E2 -22732.852} C_VEL
LIN {X 0,Y 203.555,Z 227.433,A -85,B 0,C 180,E1 -22733.463,E2 -22733.463} C_VEL
LIN {X 0,Y 201.533,Z 239.738,A -85,B 0,C 180,E1 -22734.413,E2 -22734.413} C_VEL
LIN {X 0,Y 198.708,Z 252.447,A -85,B 0,C 180,E1 -22735.842,E2 -22735.842} C_VEL
LIN {X 0,Y 196.29,Z 261.719,A -85,B 0,C 180,E1 -22737.212,E2 -22737.212} C_VEL
LIN {X 0,Y 193.575,Z 270.659,A -85,B 0,C 180,E1 -22738.844,E2 -22738.844} C_VEL
LIN {X 0,Y 190.784,Z 279.185,A -85,B 0,C 180,E1 -22740.784,E2 -22740.784} C_VEL
LIN {X 0,Y 188.166,Z 286.399,A -85,B 0,C 180,E1 -22742.772,E2 -22742.772} C_VEL
LIN {X 0,Y 185.849,Z 292.599,A -85,B 0,C 180,E1 -22744.822,E2 -22744.822} C_VEL
LIN {X 0,Y 183.432,Z 299.14,A -85,B 0,C 180,E1 -22747.472,E2 -22747.472} C_VEL
LIN {X 0,Y 181.59,Z 303.639,A -85,B 0,C 180,E1 -22749.615,E2 -22749.615} C_VEL
LIN {X 0,Y 179.359,Z 309.131,A -85,B 0,C 180,E1 -22752.91,E2 -22752.91} C_VEL
LIN {X 0,Y 177.736,Z 313.459,A -85,B 0,C 180,E1 -22756.276,E2 -22756.276} C_VEL
LIN {X 0,Y 176.984,Z 315.83,A -85,B 0,C 180,E1 -22758.548,E2 -22758.548} C_VEL
LIN {X 0,Y 176.261,Z 318.342,A -85,B 0,C 180,E1 -22761.997,E2 -22761.997} C_VEL
LIN {X 0,Y 175.394,Z 319.431,A -85,B 0,C 180,E1 -22763.871,E2 -22763.871} C_VEL
LIN {X 0,Y 173.707,Z 320.141,A -85,B 0,C 180,E1 -22765.728,E2 -22765.728} C_VEL
LIN {X 0,Y 169.956,Z 320.679,A -85,B 0,C 180,E1 -22769.525,E2 -22769.525} C_VEL
LIN {X 0,Y 168.878,Z 320.613,A -85,B 0,C 180,E1 -22771.858,E2 -22771.858} C_VEL
LIN {X 0,Y 168.86,Z 320.506,A -85,B 0,C 180,E1 -22772.196,E2 -22772.196} C_VEL
LIN {X 0,Y 168.868,Z 319.899,A -85,B 0,C 180,E1 -22774.775,E2 -22774.775} C_VEL
LIN {X 0,Y 169.417,Z 317.442,A -85,B 0,C 180,E1 -22779.551,E2 -22779.551} C_VEL
LIN {X 0,Y 170.367,Z 314.486,A -85,B 0,C 180,E1 -22783.114,E2 -22783.114} C_VEL
LIN {X 0,Y 171.854,Z 310.492,A -85,B 0,C 180,E1 -22786.634,E2 -22786.634} C_VEL
LIN {X 0,Y 174.122,Z 305.365,A -85,B 0,C 180,E1 -22790.065,E2 -22790.065} C_VEL
LIN {X 0,Y 176.392,Z 300.104,A -85,B 0,C 180,E1 -22792.859,E2 -22792.859} C_VEL
LIN {X 0,Y 178.938,Z 293.786,A -85,B 0,C 180,E1 -22795.597,E2 -22795.597} C_VEL
LIN {X 0,Y 181.249,Z 287.835,A -85,B 0,C 180,E1 -22797.73,E2 -22797.73} C_VEL
LIN {X 0,Y 183.904,Z 280.912,A -85,B 0,C 180,E1 -22799.789,E2 -22799.789} C_VEL
LIN {X 0,Y 186.801,Z 272.737,A -85,B 0,C 180,E1 -22801.784,E2 -22801.784} C_VEL
LIN {X 0,Y 189.561,Z 264.231,A -85,B 0,C 180,E1 -22803.469,E2 -22803.469} C_VEL
LIN {X 0,Y 192.015,Z 255.519,A -85,B 0,C 180,E1 -22804.882,E2 -22804.882} C_VEL
LIN {X 0,Y 194.442,Z 245.766,A -85,B 0,C 180,E1 -22806.129,E2 -22806.129} C_VEL
LIN {X 0,Y 196.492,Z 235.688,A -85,B 0,C 180,E1 -22807.126,E2 -22807.126} C_VEL
LIN {X 0,Y 198.031,Z 225.866,A -85,B 0,C 180,E1 -22807.857,E2 -22807.857} C_VEL
LIN {X 0,Y 199.134,Z 216.252,A -85,B 0,C 180,E1 -22808.361,E2 -22808.361} C_VEL
LIN {X 0,Y 201.449,Z 174.352,A -85,B 0,C 180,E1 -22809.804,E2 -22809.804} C_VEL
LIN {X 0,Y 199.678,Z 162.792,A -85,B 0,C 180,E1 -22810.76,E2 -22810.76} C_VEL
LIN {X 0,Y 193.581,Z 148.033,A -85,B 0,C 180,E1 -22813.051,E2 -22813.051} C_VEL
LIN {X 0,Y 188.724,Z 137.94,A -85,B 0,C 180,E1 -22814.962,E2 -22814.962} C_VEL
LIN {X 0,Y 181.502,Z 124.867,A -85,B 0,C 180,E1 -22818.02,E2 -22818.02} C_VEL
LIN {X 0,Y 177.619,Z 118.82,A -85,B 0,C 180,E1 -22819.79,E2 -22819.79} C_VEL
LIN {X 0,Y 174.865,Z 114.405,A -85,B 0,C 180,E1 -22821.144,E2 -22821.144} C_VEL
LIN {X 0,Y 172.025,Z 110.8,A -85,B 0,C 180,E1 -22822.574,E2 -22822.574} C_VEL
LIN {X 0,Y 171.464,Z 109.156,A -85,B 0,C 180,E1 -22823.168,E2 -22823.168} C_VEL
LIN {X 0,Y 171.395,Z 108.621,A -85,B 0,C 180,E1 -22824.244,E2 -22824.244} C_VEL
LIN {X 0,Y 171.458,Z 108.627,A -85,B 0,C 180,E1 -22829.404,E2 -22829.404} C_VEL
LIN {X 0,Y 171.464,Z 108.592,A -85,B 0,C 180,E1 -22834.388,E2 -22834.388} C_VEL
LIN {X 0,Y 171.581,Z 108.561,A -85,B 0,C 180,E1 -22840.871,E2 -22840.871} C_VEL
LIN {X 0,Y 171.612,Z 108.605,A -85,B 0,C 180,E1 -22845.775,E2 -22845.775} C_VEL
LIN {X 0,Y 171.875,Z 108.52,A -85,B 0,C 180,E1 -22850.585,E2 -22850.585} C_VEL
LIN {X 0,Y 171.825,Z 108.582,A -85,B 0,C 180,E1 -22855.306,E2 -22855.306} C_VEL
LIN {X 0,Y 172.332,Z 108.463,A -85,B 0,C 180,E1 -22859.999,E2 -22859.999} C_VEL
LIN {X 0,Y 171.824,Z 108.582,A -85,B 0,C 180,E1 -22864.691,E2 -22864.691} C_VEL
LIN {X 0,Y 171.874,Z 108.522,A -85,B 0,C 180,E1 -22869.412,E2 -22869.412} C_VEL
LIN {X 0,Y 171.611,Z 108.609,A -85,B 0,C 180,E1 -22874.223,E2 -22874.223} C_VEL
LIN {X 0,Y 171.543,Z 108.57,A -85,B 0,C 180,E1 -22879.56,E2 -22879.56} C_VEL
LIN {X 0,Y 171.467,Z 108.596,A -85,B 0,C 180,E1 -22885.615,E2 -22885.615} C_VEL
LIN {X 0,Y 171.454,Z 108.625,A -85,B 0,C 180,E1 -22890.594,E2 -22890.594} C_VEL
LIN {X 0,Y 171.41,Z 108.672,A -85,B 0,C 180,E1 -22896.705,E2 -22896.705} C_VEL
LIN {X 0,Y 171.571,Z 109.519,A -85,B 0,C 180,E1 -22897.446,E2 -22897.446} C_VEL
LIN {X 0,Y 173.114,Z 112.445,A -85,B 0,C 180,E1 -22898.385,E2 -22898.385} C_VEL
LIN {X 0,Y 175.168,Z 114.398,A -85,B 0,C 180,E1 -22899.355,E2 -22899.355} C_VEL
LIN {X 0,Y 177.261,Z 117.668,A -85,B 0,C 180,E1 -22900.38,E2 -22900.38} C_VEL
LIN {X 0,Y 178.664,Z 119.307,A -85,B 0,C 180,E1 -22901.009,E2 -22901.009} C_VEL
LIN {X 0,Y 184.811,Z 128.218,A -85,B 0,C 180,E1 -22903.664,E2 -22903.664} C_VEL
LIN {X 0,Y 190.975,Z 137.731,A -85,B 0,C 180,E1 -22906.071,E2 -22906.071} C_VEL
